//     Drive/Inputs/In/nState1 @bit 5 <-> DCM Status Channel 2/Status/Moving negative
//     Drive/Inputs/In/nState1 @bit 4 <-> DCM Status Channel 1/Status/Moving positive
//     Drive/Inputs/In/nState1 @bit 4 <-> DCM Status Channel 2/Status/Moving positive
//     Drive/Inputs/In/nState1 @bit 1 <-> DCM Status Channel 1/Status/Ready
//     Drive/Inputs/In/nState1 @bit 1 <-> DCM Status Channel 2/Status/Ready
//     Drive/Inputs/In/nState1 <-> DCM Status Channel 1/Status/Ready to enable
//     Drive/Inputs/In/nState1 <-> DCM Status Channel 2/Status/Ready to enable
//     Drive/Inputs/In/nState1 @bit 6 <-> DCM Status Channel 1/Status/Torque reduced
//     Drive/Inputs/In/nState1 @bit 6 <-> DCM Status Channel 2/Status/Torque reduced
//     Drive/Inputs/In/nState1 @bit 2 <-> DCM Status Channel 1/Status/Warning
//     Drive/Inputs/In/nState1 @bit 2 <-> DCM Status Channel 2/Status/Warning
//     Drive/Inputs/In/nState2 @bit 3 <-> DCM Status Channel 1/Status/Digital input 1
//     Drive/Inputs/In/nState2 @bit 4 <-> DCM Status Channel 1/Status/Digital input 2
//     Drive/Inputs/In/nState2 @bit 3 <-> DCM Status Channel 2/Status/Digital input 1
//     Drive/Inputs/In/nState2 @bit 4 <-> DCM Status Channel 2/Status/Digital input 2
//     Drive/Inputs/In/nState2 @bit 5 <-> DCM Status Channel 1/Status/Sync error
//     Drive/Inputs/In/nState2 @bit 5 <-> DCM Status Channel 2/Status/Sync error
//     Drive/Inputs/In/nState2 @bit 7 <-> DCM Status Channel 1/Status/TxPDO Toggle
//     Drive/Inputs/In/nState2 @bit 7 <-> DCM Status Channel 2/Status/TxPDO Toggle
//     Drive/Inputs/In/nState4 @bit 1 <-> WcState/InputToggle
//     Drive/Inputs/In/nState4 <-> WcState/WcState
//     Drive/Outputs/Out/nCtrl1 <-> DCM Control Channel 1/Control/Enable
//     Drive/Outputs/Out/nCtrl1 <-> DCM Control Channel 2/Control/Enable
//     Drive/Outputs/Out/nCtrl1 @bit 2 <-> DCM Control Channel 1/Control/Reduce torque
//     Drive/Outputs/Out/nCtrl1 @bit 2 <-> DCM Control Channel 2/Control/Reduce torque
//     Drive/Outputs/Out/nCtrl1 @bit 1 <-> DCM Control Channel 1/Control/Reset
//     Drive/Outputs/Out/nCtrl1 @bit 1 <-> DCM Control Channel 2/Control/Reset
//     Drive/Outputs/Out/nDataOut2[0] <-> DCM Velocity Channel 1/Velocity
//     Drive/Outputs/Out/nDataOut2[0] <-> DCM Velocity Channel 2/Velocity
//     Enc/Inputs/In/nDataIn1[0] <-> ENC Status compact Channel 1/Counter value
//     Enc/Inputs/In/nDataIn1[0] <-> ENC Status compact Channel 2/Counter value
//     Enc/Inputs/In/nDataIn2[0] <-> ENC Status compact Channel 1/Latch value
//     Enc/Inputs/In/nDataIn2[0] <-> ENC Status compact Channel 2/Latch value
//     Enc/Inputs/In/nState1 @bit 4 <-> ENC Status compact Channel 1/Status/Counter overflow
//     Enc/Inputs/In/nState1 @bit 4 <-> ENC Status compact Channel 2/Status/Counter overflow
//     Enc/Inputs/In/nState1 @bit 3 <-> ENC Status compact Channel 1/Status/Counter underflow
//     Enc/Inputs/In/nState1 @bit 3 <-> ENC Status compact Channel 2/Status/Counter underflow
//     Enc/Inputs/In/nState1 @bit 7 <-> ENC Status compact Channel 1/Status/Extrapolation stall
//     Enc/Inputs/In/nState1 @bit 7 <-> ENC Status compact Channel 2/Status/Extrapolation stall
//     Enc/Inputs/In/nState1 @bit 1 <-> ENC Status compact Channel 1/Status/Latch extern valid
//     Enc/Inputs/In/nState1 @bit 1 <-> ENC Status compact Channel 2/Status/Latch extern valid
//     Enc/Inputs/In/nState1 @bit 2 <-> ENC Status compact Channel 1/Status/Set counter done
//     Enc/Inputs/In/nState1 @bit 2 <-> ENC Status compact Channel 2/Status/Set counter done
//     Enc/Inputs/In/nState2 @bit 4 <-> ENC Status compact Channel 1/Status/Status of extern latch
//     Enc/Inputs/In/nState2 @bit 4 <-> ENC Status compact Channel 2/Status/Status of extern latch
//     Enc/Inputs/In/nState2 <-> ENC Status compact Channel 1/Status/Status of input A
//     Enc/Inputs/In/nState2 <-> ENC Status compact Channel 2/Status/Status of input A
//     Enc/Inputs/In/nState2 @bit 1 <-> ENC Status compact Channel 1/Status/Status of input B
//     Enc/Inputs/In/nState2 @bit 1 <-> ENC Status compact Channel 2/Status/Status of input B
//     Enc/Inputs/In/nState2 @bit 5 <-> ENC Status compact Channel 1/Status/Sync error
//     Enc/Inputs/In/nState2 @bit 5 <-> ENC Status compact Channel 2/Status/Sync error
//     Enc/Inputs/In/nState2 @bit 7 <-> ENC Status compact Channel 1/Status/TxPDO Toggle
//     Enc/Inputs/In/nState2 @bit 7 <-> ENC Status compact Channel 2/Status/TxPDO Toggle
//     Enc/Inputs/In/nState4 @bit 1 <-> WcState/InputToggle
//     Enc/Inputs/In/nState4 <-> WcState/WcState
//     Enc/Outputs/Out/nCtrl1 @bit 3 <-> ENC Control compact Channel 1/Control/Enable latch extern on negative edge
//     Enc/Outputs/Out/nCtrl1 @bit 3 <-> ENC Control compact Channel 2/Control/Enable latch extern on negative edge
//     Enc/Outputs/Out/nCtrl1 @bit 1 <-> ENC Control compact Channel 1/Control/Enable latch extern on positive edge
//     Enc/Outputs/Out/nCtrl1 @bit 1 <-> ENC Control compact Channel 2/Control/Enable latch extern on positive edge
//     Enc/Outputs/Out/nCtrl1 @bit 2 <-> ENC Control compact Channel 1/Control/Set counter
//     Enc/Outputs/Out/nCtrl1 @bit 2 <-> ENC Control compact Channel 2/Control/Set counter
//     Enc/Outputs/Out/nDataOut1[0] <-> ENC Control compact Channel 1/Set counter value
//     Enc/Outputs/Out/nDataOut1[0] <-> ENC Control compact Channel 2/Set counter value
//   (this object) <-> Device 1 (EtherCAT)/Power (EK1200)/PLC Junction 3 (EK1122)/X1 TMO FEE EC1 (EK1100)/TMO FEE EC1 E1 (EK1122)/X2-ST1K4-TEST (EK1100)/ST1K4-EL5042-E6
//     Enc/Inputs/In/nComState @bit 1 <-> WcState/InputToggle
//     Enc/Inputs/In/nComState <-> WcState/WcState
//     Enc/Inputs/In/nDataIn1 <-> FB Inputs Channel 1/Position
//     Enc/Inputs/In/nState1 @bit 12 <-> FB Inputs Channel 1/Status/Diag
//     Enc/Inputs/In/nState1 @bit 1 <-> FB Inputs Channel 1/Status/Error
//     Enc/Inputs/In/nState1 @bit 14 <-> FB Inputs Channel 1/Status/Input cycle counter
//     Enc/Inputs/In/nState1 @bit 2 <-> FB Inputs Channel 1/Status/Ready
//     Enc/Inputs/In/nState1 @bit 13 <-> FB Inputs Channel 1/Status/TxPDO State
//     Enc/Inputs/In/nState1 <-> FB Inputs Channel 1/Status/Warning
//   (this object) <-> Device 1 (EtherCAT)/Power (EK1200)/PLC Junction 3 (EK1122)/X1 TMO FEE EC1 (EK1100)/TMO FEE EC1 E1 (EK1122)/X2-ST1K4-TEST (EK1100)/ST1K4-EL7041-E4
//     Drive/Inputs/In/nState1 @bit 3 <-> STM Status/Status/Error
//     Drive/Inputs/In/nState1 @bit 5 <-> STM Status/Status/Moving negative
//     Drive/Inputs/In/nState1 @bit 4 <-> STM Status/Status/Moving positive
//     Drive/Inputs/In/nState1 @bit 1 <-> STM Status/Status/Ready
//     Drive/Inputs/In/nState1 <-> STM Status/Status/Ready to enable
//     Drive/Inputs/In/nState1 @bit 6 <-> STM Status/Status/Torque reduced
//     Drive/Inputs/In/nState1 @bit 2 <-> STM Status/Status/Warning
//     Drive/Inputs/In/nState2 @bit 3 <-> STM Status/Status/Digital input 1
//     Drive/Inputs/In/nState2 @bit 4 <-> STM Status/Status/Digital input 2
//     Drive/Inputs/In/nState2 @bit 5 <-> STM Status/Status/Sync error
//     Drive/Inputs/In/nState2 @bit 7 <-> STM Status/Status/TxPDO Toggle
//     Drive/Inputs/In/nState4 @bit 1 <-> WcState/InputToggle
//     Drive/Inputs/In/nState4 <-> WcState/WcState
//     Drive/Outputs/Out/nCtrl1 <-> STM Control/Control/Enable
//     Drive/Outputs/Out/nCtrl1 @bit 2 <-> STM Control/Control/Reduce torque
//     Drive/Outputs/Out/nCtrl1 @bit 1 <-> STM Control/Control/Reset
//     Drive/Outputs/Out/nDataOut2[0] <-> STM Velocity/Velocity
//   kfe_motion Instance <-> Device 1 (EtherCAT)/Power (EK1200)/PLC Junction 1 (EK1122)/X1 RTDSK0 (EK1100)/RTDSK0-EL2004
//     PlcTask Outputs/PRG_RTDSK0.bRTDSK0_SCRP_LED_01 <-> Channel 3/Output
//   kfe_motion Instance <-> Device 1 (EtherCAT)/Power (EK1200)/PLC Junction 1 (EK1122)/X1 RTDSK0 (EK1100)/RTDSK0-M2-EL7041
//     PlcTask Inputs/Main.M11.bLimitBackwardEnable <-> STM Status/Status/Digital input 2
//     PlcTask Inputs/Main.M11.bLimitForwardEnable <-> STM Status/Status/Digital input 1
//   kfe_motion Instance <-> Device 1 (EtherCAT)/Power (EK1200)/PLC Junction 1 (EK1122)/X1 RTDSK0 (EK1100)/RTDSK0-M3-EL7041
//     PlcTask Inputs/Main.M12.bLimitBackwardEnable <-> STM Status/Status/Digital input 2
//     PlcTask Inputs/Main.M12.bLimitForwardEnable <-> STM Status/Status/Digital input 1
//   kfe_motion Instance <-> Device 1 (EtherCAT)/Power (EK1200)/PLC Junction 1 (EK1122)/X1 RTDSK0 (EK1100)/RTDSK0-M4-EL7041
//     PlcTask Inputs/Main.M13.bLimitBackwardEnable <-> STM Status/Status/Digital input 2
//     PlcTask Inputs/Main.M13.bLimitForwardEnable <-> STM Status/Status/Digital input 1
//   kfe_motion Instance <-> Device 1 (EtherCAT)/Power (EK1200)/PLC Junction 1 (EK1122)/X1 RTDSK0 (EK1100)/RTDSK0-MPA-EL1008
//     PlcTask Inputs/PRG_RTDSK0.RTDSK0_MPA_01.i_xInsertedLS <-> Channel 1/Input
//     PlcTask Inputs/PRG_RTDSK0.RTDSK0_MPA_02.i_xInsertedLS <-> Channel 3/Input
//     PlcTask Inputs/PRG_RTDSK0.RTDSK0_MPA_03.i_xInsertedLS <-> Channel 5/Input
//     PlcTask Inputs/PRG_RTDSK0.RTDSK0_MPA_04.i_xInsertedLS <-> Channel 7/Input
//     PlcTask Inputs/PRG_RTDSK0.RTDSK0_MPA_01.i_xRetractedLS <-> Channel 2/Input
//     PlcTask Inputs/PRG_RTDSK0.RTDSK0_MPA_02.i_xRetractedLS <-> Channel 4/Input
//     PlcTask Inputs/PRG_RTDSK0.RTDSK0_MPA_03.i_xRetractedLS <-> Channel 6/Input
//     PlcTask Inputs/PRG_RTDSK0.RTDSK0_MPA_04.i_xRetractedLS <-> Channel 8/Input
//   kfe_motion Instance <-> Device 1 (EtherCAT)/Power (EK1200)/PLC Junction 1 (EK1122)/X1 RTDSK0 (EK1100)/RTDSK0-MPA-EL2008
//     PlcTask Outputs/PRG_RTDSK0.RTDSK0_MPA_01.q_xInsert_DO <-> Channel 1/Output
//     PlcTask Outputs/PRG_RTDSK0.RTDSK0_MPA_02.q_xInsert_DO <-> Channel 3/Output
//     PlcTask Outputs/PRG_RTDSK0.RTDSK0_MPA_03.q_xInsert_DO <-> Channel 5/Output
//     PlcTask Outputs/PRG_RTDSK0.RTDSK0_MPA_04.q_xInsert_DO <-> Channel 7/Output
//     PlcTask Outputs/PRG_RTDSK0.RTDSK0_MPA_01.q_xRetract_DO <-> Channel 2/Output
//     PlcTask Outputs/PRG_RTDSK0.RTDSK0_MPA_02.q_xRetract_DO <-> Channel 4/Output
//     PlcTask Outputs/PRG_RTDSK0.RTDSK0_MPA_03.q_xRetract_DO <-> Channel 6/Output
//     PlcTask Outputs/PRG_RTDSK0.RTDSK0_MPA_04.q_xRetract_DO <-> Channel 8/Output
//   kfe_motion Instance <-> Device 1 (EtherCAT)/Power (EK1200)/PLC Junction 1 (EK1122)/X2 IM1K0-XTES (EK1100)/IM1K0-EL1004
//     PlcTask Inputs/PRG_IM1K0_XTES.fbIM1K0.fbFlowSwitch.bFlowOk <-> Channel 2/Input
//     PlcTask Inputs/PRG_OTHER.fbPC1K0FlowSwitch.bFlowOk <-> Channel 1/Input
//     PlcTask Inputs/PRG_SL1K0_POWER.fbSL1K0.fbFlowSwitch.bFlowOk <-> Channel 3/Input
//   kfe_motion Instance <-> Device 1 (EtherCAT)/Power (EK1200)/PLC Junction 1 (EK1122)/X2 IM1K0-XTES (EK1100)/IM1K0-EL1088
//     PlcTask Inputs/Main.M2.bHome <-> Channel 2/Input
//     PlcTask Inputs/Main.M3.bHome <-> Channel 4/Input
//     PlcTask Inputs/PRG_IM1K0_XTES.fbIM1K0.bFocusEndBwd <-> Channel 4/Input
//     PlcTask Inputs/PRG_IM1K0_XTES.fbIM1K0.bFocusEndFwd <-> Channel 3/Input
//     PlcTask Inputs/PRG_IM1K0_XTES.fbIM1K0.bZoomEndBwd <-> Channel 2/Input
//     PlcTask Inputs/PRG_IM1K0_XTES.fbIM1K0.bZoomEndFwd <-> Channel 1/Input
//   kfe_motion Instance <-> Device 1 (EtherCAT)/Power (EK1200)/PLC Junction 1 (EK1122)/X2 IM1K0-XTES (EK1100)/IM1K0-EL2004
//     PlcTask Outputs/Main.M1.bBrakeRelease <-> Channel 1/Output
//     PlcTask Outputs/PRG_IM1K0_XTES.fbIM1K0.fbLED.bLEDPower <-> Channel 3/Output
//     PlcTask Outputs/PRG_IM1K0_XTES.fbIM1K0.fbOpal.bOpalPower <-> Channel 2/Output
//   kfe_motion Instance <-> Device 1 (EtherCAT)/Power (EK1200)/PLC Junction 1 (EK1122)/X2 IM1K0-XTES (EK1100)/IM1K0-EL3054
//     PlcTask Inputs/Main.M1.nRawEncoderINT <-> AI Standard Channel 1/Value
//   kfe_motion Instance <-> Device 1 (EtherCAT)/Power (EK1200)/PLC Junction 1 (EK1122)/X2 IM1K0-XTES (EK1100)/IM1K0-EL5101-01
//     PlcTask Inputs/Main.M2.nRawEncoderUINT <-> ENC Status compact/Counter value
//     PlcTask Inputs/Main.M3.nRawEncoderUINT <-> ENC Status compact/Counter value
//   kfe_motion Instance <-> Device 1 (EtherCAT)/Power (EK1200)/PLC Junction 1 (EK1122)/X2 IM1K0-XTES (EK1100)/IM1K0-EL6002
//     PlcTask Inputs/PRG_IM1K0_XTES.stEL6In/D[{0..21}] <-> COM TxPDO-Map Inputs Channel 1/Data In {0..21}  (22 links)
//     PlcTask Inputs/PRG_IM1K0_XTES.stEL6In/Status <-> COM TxPDO-Map Inputs Channel 1/Status
//     PlcTask Outputs/PRG_IM1K0_XTES.stEL6Out/Ctrl <-> COM RxPDO-Map Outputs Channel 1/Ctrl
//     PlcTask Outputs/PRG_IM1K0_XTES.stEL6Out/D[{0..21}] <-> COM RxPDO-Map Outputs Channel 1/Data Out {0..21}  (22 links)
//   kfe_motion Instance <-> Device 1 (EtherCAT)/Power (EK1200)/PLC Junction 1 (EK1122)/X2 IM1K0-XTES (EK1100)/IM1K0-EL7041
//     PlcTask Inputs/Main.M1.bLimitForwardEnable <-> STM Status/Status/Digital input 1
//   kfe_motion Instance <-> Device 1 (EtherCAT)/Power (EK1200)/PLC Junction 2 (EK1122)/X1 SL1K0-POWER (EK1100)/SL1K0-EL3054-E12
//     PlcTask Inputs/Main.M{18..21}.nRawEncoderINT <-> AI Standard Channel {1..4}/Value  (4 links)
//   kfe_motion Instance <-> Device 1 (EtherCAT)/Power (EK1200)/PLC Junction 2 (EK1122)/X1 SL1K0-POWER (EK1100)/SL1K0-EL3202-E6
//     PlcTask Inputs/PRG_SL1K0_POWER.fbSL1K0.RTD_South_1.bError <-> RTD Inputs Channel 1/Status/Error
//     PlcTask Inputs/PRG_SL1K0_POWER.fbSL1K0.RTD_South_2.bError <-> RTD Inputs Channel 2/Status/Error
//     PlcTask Inputs/PRG_SL1K0_POWER.fbSL1K0.RTD_South_1.bOverrange <-> RTD Inputs Channel 1/Status/Overrange
//     PlcTask Inputs/PRG_SL1K0_POWER.fbSL1K0.RTD_South_2.bOverrange <-> RTD Inputs Channel 2/Status/Overrange
//     PlcTask Inputs/PRG_SL1K0_POWER.fbSL1K0.RTD_South_1.bUnderrange <-> RTD Inputs Channel 1/Status/Underrange
//     PlcTask Inputs/PRG_SL1K0_POWER.fbSL1K0.RTD_South_2.bUnderrange <-> RTD Inputs Channel 2/Status/Underrange
//     PlcTask Inputs/PRG_SL1K0_POWER.fbSL1K0.RTD_South_1.iRaw <-> RTD Inputs Channel 1/Value
//     PlcTask Inputs/PRG_SL1K0_POWER.fbSL1K0.RTD_South_2.iRaw <-> RTD Inputs Channel 2/Value
//   kfe_motion Instance <-> Device 1 (EtherCAT)/Power (EK1200)/PLC Junction 2 (EK1122)/X1 SL1K0-POWER (EK1100)/SL1K0-EL3202-E7
//     PlcTask Inputs/PRG_SL1K0_POWER.fbSL1K0.RTD_TOP_1.bError <-> RTD Inputs Channel 1/Status/Error
//     PlcTask Inputs/PRG_SL1K0_POWER.fbSL1K0.RTD_TOP_2.bError <-> RTD Inputs Channel 2/Status/Error
//     PlcTask Inputs/PRG_SL1K0_POWER.fbSL1K0.RTD_TOP_1.bOverrange <-> RTD Inputs Channel 1/Status/Overrange
//     PlcTask Inputs/PRG_SL1K0_POWER.fbSL1K0.RTD_TOP_2.bOverrange <-> RTD Inputs Channel 2/Status/Overrange
//     PlcTask Inputs/PRG_SL1K0_POWER.fbSL1K0.RTD_TOP_1.bUnderrange <-> RTD Inputs Channel 1/Status/Underrange
//     PlcTask Inputs/PRG_SL1K0_POWER.fbSL1K0.RTD_TOP_2.bUnderrange <-> RTD Inputs Channel 2/Status/Underrange
//     PlcTask Inputs/PRG_SL1K0_POWER.fbSL1K0.RTD_TOP_1.iRaw <-> RTD Inputs Channel 1/Value
//     PlcTask Inputs/PRG_SL1K0_POWER.fbSL1K0.RTD_TOP_2.iRaw <-> RTD Inputs Channel 2/Value
//   kfe_motion Instance <-> Device 1 (EtherCAT)/Power (EK1200)/PLC Junction 2 (EK1122)/X1 SL1K0-POWER (EK1100)/SL1K0-EL3202-E8
//     PlcTask Inputs/PRG_SL1K0_POWER.fbSL1K0.RTD_North_1.bError <-> RTD Inputs Channel 1/Status/Error
//     PlcTask Inputs/PRG_SL1K0_POWER.fbSL1K0.RTD_North_2.bError <-> RTD Inputs Channel 2/Status/Error
//     PlcTask Inputs/PRG_SL1K0_POWER.fbSL1K0.RTD_North_1.bOverrange <-> RTD Inputs Channel 1/Status/Overrange
//     PlcTask Inputs/PRG_SL1K0_POWER.fbSL1K0.RTD_North_2.bOverrange <-> RTD Inputs Channel 2/Status/Overrange
//     PlcTask Inputs/PRG_SL1K0_POWER.fbSL1K0.RTD_North_1.bUnderrange <-> RTD Inputs Channel 1/Status/Underrange
//     PlcTask Inputs/PRG_SL1K0_POWER.fbSL1K0.RTD_North_2.bUnderrange <-> RTD Inputs Channel 2/Status/Underrange
//     PlcTask Inputs/PRG_SL1K0_POWER.fbSL1K0.RTD_North_1.iRaw <-> RTD Inputs Channel 1/Value
//     PlcTask Inputs/PRG_SL1K0_POWER.fbSL1K0.RTD_North_2.iRaw <-> RTD Inputs Channel 2/Value
//   kfe_motion Instance <-> Device 1 (EtherCAT)/Power (EK1200)/PLC Junction 2 (EK1122)/X1 SL1K0-POWER (EK1100)/SL1K0-EL3202-E9
//     PlcTask Inputs/PRG_SL1K0_POWER.fbSL1K0.RTD_Bottom_1.bError <-> RTD Inputs Channel 1/Status/Error
//     PlcTask Inputs/PRG_SL1K0_POWER.fbSL1K0.RTD_Bottom_2.bError <-> RTD Inputs Channel 2/Status/Error
//     PlcTask Inputs/PRG_SL1K0_POWER.fbSL1K0.RTD_Bottom_1.bOverrange <-> RTD Inputs Channel 1/Status/Overrange
//     PlcTask Inputs/PRG_SL1K0_POWER.fbSL1K0.RTD_Bottom_2.bOverrange <-> RTD Inputs Channel 2/Status/Overrange
//     PlcTask Inputs/PRG_SL1K0_POWER.fbSL1K0.RTD_Bottom_1.bUnderrange <-> RTD Inputs Channel 1/Status/Underrange
//     PlcTask Inputs/PRG_SL1K0_POWER.fbSL1K0.RTD_Bottom_2.bUnderrange <-> RTD Inputs Channel 2/Status/Underrange
//     PlcTask Inputs/PRG_SL1K0_POWER.fbSL1K0.RTD_Bottom_1.iRaw <-> RTD Inputs Channel 1/Value
//     PlcTask Inputs/PRG_SL1K0_POWER.fbSL1K0.RTD_Bottom_2.iRaw <-> RTD Inputs Channel 2/Value
//   kfe_motion Instance <-> Device 1 (EtherCAT)/Power (EK1200)/PLC Junction 2 (EK1122)/X1 SL1K0-POWER (EK1100)/SL1K0-EL7041-E1
//     PlcTask Inputs/Main.M18.bLimitBackwardEnable <-> STM Status/Status/Digital input 1
//     PlcTask Inputs/Main.M18.bLimitForwardEnable <-> STM Status/Status/Digital input 2
//   kfe_motion Instance <-> Device 1 (EtherCAT)/Power (EK1200)/PLC Junction 2 (EK1122)/X1 SL1K0-POWER (EK1100)/SL1K0-EL7041-E2
//     PlcTask Inputs/Main.M19.bLimitBackwardEnable <-> STM Status/Status/Digital input 1
//     PlcTask Inputs/Main.M19.bLimitForwardEnable <-> STM Status/Status/Digital input 2
//   kfe_motion Instance <-> Device 1 (EtherCAT)/Power (EK1200)/PLC Junction 2 (EK1122)/X1 SL1K0-POWER (EK1100)/SL1K0-EL7041-E4
//     PlcTask Inputs/Main.M20.bLimitBackwardEnable <-> STM Status/Status/Digital input 1
//     PlcTask Inputs/Main.M20.bLimitForwardEnable <-> STM Status/Status/Digital input 2
//   kfe_motion Instance <-> Device 1 (EtherCAT)/Power (EK1200)/PLC Junction 2 (EK1122)/X1 SL1K0-POWER (EK1100)/SL1K0-EL7041-E5
//     PlcTask Inputs/Main.M21.bLimitBackwardEnable <-> STM Status/Status/Digital input 1
//     PlcTask Inputs/Main.M21.bLimitForwardEnable <-> STM Status/Status/Digital input 2
//   kfe_motion Instance <-> Device 1 (EtherCAT)/Power (EK1200)/PLC Junction 2 (EK1122)/X2 SXR EC1 (EK1100)/EC1 E1 (EK1122)/X1 IM2K0-XTES (EK1100)/IM2K0-EL1088
//     PlcTask Inputs/Main.M6.bHome <-> Channel 2/Input
//     PlcTask Inputs/Main.M7.bHome <-> Channel 4/Input
//   kfe_motion Instance <-> Device 1 (EtherCAT)/Power (EK1200)/PLC Junction 2 (EK1122)/X2 SXR EC1 (EK1100)/EC1 E1 (EK1122)/X1 IM2K0-XTES (EK1100)/IM2K0-EL2004
//     PlcTask Outputs/Main.M5.bBrakeRelease <-> Channel 1/Output
//     PlcTask Outputs/PRG_IM2K0_XTES.fbIM2K0.fbGige.bGigePower <-> Channel 4/Output
//     PlcTask Outputs/PRG_IM2K0_XTES.fbIM2K0.fbLED.bLEDPower <-> Channel 3/Output
//   kfe_motion Instance <-> Device 1 (EtherCAT)/Power (EK1200)/PLC Junction 2 (EK1122)/X2 SXR EC1 (EK1100)/EC1 E1 (EK1122)/X1 IM2K0-XTES (EK1100)/IM2K0-EL5042
//     PlcTask Inputs/Main.M5.nRawEncoderULINT <-> FB Inputs Channel 1/Position
//   kfe_motion Instance <-> Device 1 (EtherCAT)/Power (EK1200)/PLC Junction 2 (EK1122)/X2 SXR EC1 (EK1100)/EC1 E1 (EK1122)/X1 IM2K0-XTES (EK1100)/IM2K0-EL7041
//     PlcTask Inputs/PRG_IM2K0_XTES.bDefectiveLimitSwitch <-> STM Status/Status/Digital input 1
//   kfe_motion Instance <-> Device 1 (EtherCAT)/Power (EK1200)/PLC Junction 2 (EK1122)/X2 SXR EC1 (EK1100)/EC1 E1 (EK1122)/X1 IM2K0-XTES (EK1100)/IM2K0-EL7342
//     PlcTask Inputs/Main.M6.nRawEncoderUINT <-> ENC Status compact Channel 1/Counter value
//     PlcTask Inputs/Main.M7.nRawEncoderUINT <-> ENC Status compact Channel 2/Counter value
//   kfe_motion Instance <-> Device 1 (EtherCAT)/Power (EK1200)/PLC Junction 2 (EK1122)/X2 SXR EC1 (EK1100)/EC1 E1 (EK1122)/X2 SL2K0-POWER (EK1100)/SL2K0-EL1004-E12
//     PlcTask Inputs/PRG_IM2K0_XTES.fbIM2K0.fbFlowSwitch.bFlowOk <-> Channel 1/Input
//     PlcTask Inputs/PRG_PF1K0_WFS.fbPF1K0.fbFlowSwitch.bFlowOk <-> Channel 1/Input
//     PlcTask Inputs/PRG_SL2K0_POWER.fbSL2K0.fbFlowSwitch.bFlowOk <-> Channel 1/Input
//   kfe_motion Instance <-> Device 1 (EtherCAT)/Power (EK1200)/PLC Junction 2 (EK1122)/X2 SXR EC1 (EK1100)/EC1 E1 (EK1122)/X2 SL2K0-POWER (EK1100)/SL2K0-EL3202-E10
//     PlcTask Inputs/PRG_SL2K0_POWER.fbSL2K0.RTD_Bottom_1.bError <-> RTD Inputs Channel 1/Status/Error
//     PlcTask Inputs/PRG_SL2K0_POWER.fbSL2K0.RTD_Bottom_1.iRaw <-> RTD Inputs Channel 1/Value
//     PlcTask Inputs/PRG_SL2K0_POWER.fbSL2K0.RTD_North_1.bError <-> RTD Inputs Channel 1/Status/Error
//     PlcTask Inputs/PRG_SL2K0_POWER.fbSL2K0.RTD_North_2.bError <-> RTD Inputs Channel 2/Status/Error
//     PlcTask Inputs/PRG_SL2K0_POWER.fbSL2K0.RTD_North_1.bOverrange <-> RTD Inputs Channel 1/Status/Overrange
//     PlcTask Inputs/PRG_SL2K0_POWER.fbSL2K0.RTD_North_2.bOverrange <-> RTD Inputs Channel 2/Status/Overrange
//     PlcTask Inputs/PRG_SL2K0_POWER.fbSL2K0.RTD_North_1.bUnderrange <-> RTD Inputs Channel 1/Status/Underrange
//     PlcTask Inputs/PRG_SL2K0_POWER.fbSL2K0.RTD_North_2.bUnderrange <-> RTD Inputs Channel 2/Status/Underrange
//     PlcTask Inputs/PRG_SL2K0_POWER.fbSL2K0.RTD_North_1.iRaw <-> RTD Inputs Channel 1/Value
//     PlcTask Inputs/PRG_SL2K0_POWER.fbSL2K0.RTD_North_2.iRaw <-> RTD Inputs Channel 2/Value
//   kfe_motion Instance <-> Device 1 (EtherCAT)/Power (EK1200)/PLC Junction 2 (EK1122)/X2 SXR EC1 (EK1100)/EC1 E1 (EK1122)/X2 SL2K0-POWER (EK1100)/SL2K0-EL3202-E11
//     PlcTask Inputs/PRG_SL2K0_POWER.fbSL2K0.RTD_Bottom_1.bOverrange <-> RTD Inputs Channel 1/Status/Overrange
//     PlcTask Inputs/PRG_SL2K0_POWER.fbSL2K0.RTD_Bottom_2.bOverrange <-> RTD Inputs Channel 2/Status/Overrange
//     PlcTask Inputs/PRG_SL2K0_POWER.fbSL2K0.RTD_Bottom_1.bUnderrange <-> RTD Inputs Channel 1/Status/Underrange
//     PlcTask Inputs/PRG_SL2K0_POWER.fbSL2K0.RTD_Bottom_2.bUnderrange <-> RTD Inputs Channel 2/Status/Underrange
//     PlcTask Inputs/PRG_SL2K0_POWER.fbSL2K0.RTD_Bottom_2.bError <-> RTD Inputs Channel 2/Status/Error
//     PlcTask Inputs/PRG_SL2K0_POWER.fbSL2K0.RTD_Bottom_2.iRaw <-> RTD Inputs Channel 2/Value
//   kfe_motion Instance <-> Device 1 (EtherCAT)/Power (EK1200)/PLC Junction 2 (EK1122)/X2 SXR EC1 (EK1100)/EC1 E1 (EK1122)/X2 SL2K0-POWER (EK1100)/SL2K0-EL3202-E8
//     PlcTask Inputs/PRG_SL2K0_POWER.fbSL2K0.RTD_South_1.bError <-> RTD Inputs Channel 1/Status/Error
//     PlcTask Inputs/PRG_SL2K0_POWER.fbSL2K0.RTD_South_2.bError <-> RTD Inputs Channel 2/Status/Error
//     PlcTask Inputs/PRG_SL2K0_POWER.fbSL2K0.RTD_South_1.bOverrange <-> RTD Inputs Channel 1/Status/Overrange
//     PlcTask Inputs/PRG_SL2K0_POWER.fbSL2K0.RTD_South_2.bOverrange <-> RTD Inputs Channel 2/Status/Overrange
//     PlcTask Inputs/PRG_SL2K0_POWER.fbSL2K0.RTD_South_1.bUnderrange <-> RTD Inputs Channel 1/Status/Underrange
//     PlcTask Inputs/PRG_SL2K0_POWER.fbSL2K0.RTD_South_2.bUnderrange <-> RTD Inputs Channel 2/Status/Underrange
//     PlcTask Inputs/PRG_SL2K0_POWER.fbSL2K0.RTD_South_1.iRaw <-> RTD Inputs Channel 1/Value
//     PlcTask Inputs/PRG_SL2K0_POWER.fbSL2K0.RTD_South_2.iRaw <-> RTD Inputs Channel 2/Value
//   kfe_motion Instance <-> Device 1 (EtherCAT)/Power (EK1200)/PLC Junction 2 (EK1122)/X2 SXR EC1 (EK1100)/EC1 E1 (EK1122)/X2 SL2K0-POWER (EK1100)/SL2K0-EL3202-E9
//     PlcTask Inputs/PRG_SL2K0_POWER.fbSL2K0.RTD_TOP_1.bError <-> RTD Inputs Channel 1/Status/Error
//     PlcTask Inputs/PRG_SL2K0_POWER.fbSL2K0.RTD_TOP_2.bError <-> RTD Inputs Channel 2/Status/Error
//     PlcTask Inputs/PRG_SL2K0_POWER.fbSL2K0.RTD_TOP_1.bOverrange <-> RTD Inputs Channel 1/Status/Overrange
//     PlcTask Inputs/PRG_SL2K0_POWER.fbSL2K0.RTD_TOP_2.bOverrange <-> RTD Inputs Channel 2/Status/Overrange
//     PlcTask Inputs/PRG_SL2K0_POWER.fbSL2K0.RTD_TOP_1.bUnderrange <-> RTD Inputs Channel 1/Status/Underrange
//     PlcTask Inputs/PRG_SL2K0_POWER.fbSL2K0.RTD_TOP_2.bUnderrange <-> RTD Inputs Channel 2/Status/Underrange
//     PlcTask Inputs/PRG_SL2K0_POWER.fbSL2K0.RTD_TOP_1.iRaw <-> RTD Inputs Channel 1/Value
//     PlcTask Inputs/PRG_SL2K0_POWER.fbSL2K0.RTD_TOP_2.iRaw <-> RTD Inputs Channel 2/Value
//   kfe_motion Instance <-> Device 1 (EtherCAT)/Power (EK1200)/PLC Junction 2 (EK1122)/X2 SXR EC1 (EK1100)/EC1 E1 (EK1122)/X2 SL2K0-POWER (EK1100)/SL2K0-EL5042-E2
//     PlcTask Inputs/Main.M22.nRawEncoderUINT <-> FB Inputs Channel 1/Position
//     PlcTask Inputs/Main.M23.nRawEncoderUINT <-> FB Inputs Channel 2/Position
//   kfe_motion Instance <-> Device 1 (EtherCAT)/Power (EK1200)/PLC Junction 2 (EK1122)/X2 SXR EC1 (EK1100)/EC1 E1 (EK1122)/X2 SL2K0-POWER (EK1100)/SL2K0-EL5042-E6
//     PlcTask Inputs/Main.M24.nRawEncoderUINT <-> FB Inputs Channel 1/Position
//     PlcTask Inputs/Main.M25.nRawEncoderUINT <-> FB Inputs Channel 2/Position
//   kfe_motion Instance <-> Device 1 (EtherCAT)/Power (EK1200)/PLC Junction 2 (EK1122)/X2 SXR EC1 (EK1100)/EC1 E1 (EK1122)/X2 SL2K0-POWER (EK1100)/SL2K0-EL7041-E1
//     PlcTask Inputs/Main.M22.bLimitBackwardEnable <-> STM Status/Status/Digital input 1
//     PlcTask Inputs/Main.M22.bLimitForwardEnable <-> STM Status/Status/Digital input 2
//   kfe_motion Instance <-> Device 1 (EtherCAT)/Power (EK1200)/PLC Junction 2 (EK1122)/X2 SXR EC1 (EK1100)/EC1 E1 (EK1122)/X2 SL2K0-POWER (EK1100)/SL2K0-EL7041-E3
//     PlcTask Inputs/Main.M23.bLimitBackwardEnable <-> STM Status/Status/Digital input 1
//     PlcTask Inputs/Main.M23.bLimitForwardEnable <-> STM Status/Status/Digital input 2
//   kfe_motion Instance <-> Device 1 (EtherCAT)/Power (EK1200)/PLC Junction 2 (EK1122)/X2 SXR EC1 (EK1100)/EC1 E1 (EK1122)/X2 SL2K0-POWER (EK1100)/SL2K0-EL7041-E5
//     PlcTask Inputs/Main.M24.bLimitBackwardEnable <-> STM Status/Status/Digital input 1
//     PlcTask Inputs/Main.M24.bLimitForwardEnable <-> STM Status/Status/Digital input 2
//   kfe_motion Instance <-> Device 1 (EtherCAT)/Power (EK1200)/PLC Junction 2 (EK1122)/X2 SXR EC1 (EK1100)/EC1 E1 (EK1122)/X2 SL2K0-POWER (EK1100)/SL2K0-EL7041-E7
//     PlcTask Inputs/Main.M25.bLimitBackwardEnable <-> STM Status/Status/Digital input 1
//     PlcTask Inputs/Main.M25.bLimitForwardEnable <-> STM Status/Status/Digital input 2
//   kfe_motion Instance <-> Device 1 (EtherCAT)/Power (EK1200)/PLC Junction 2 (EK1122)/X2 SXR EC1 (EK1100)/EC1 E2 (EK1122)/X1 PF1K0-WFS (EK1100)/PF1K0-EL2004
//     PlcTask Outputs/Main.M8.bBrakeRelease <-> Channel 1/Output
//   kfe_motion Instance <-> Device 1 (EtherCAT)/Power (EK1200)/PLC Junction 2 (EK1122)/X2 SXR EC1 (EK1100)/EC1 E2 (EK1122)/X1 PF1K0-WFS (EK1100)/PF1K0-EL3062
//     PlcTask Inputs/PRG_PF1K0_PM.fbPowerMeter.iVoltageINT <-> AI Standard Channel 1/Value
//   kfe_motion Instance <-> Device 1 (EtherCAT)/Power (EK1200)/PLC Junction 2 (EK1122)/X2 SXR EC1 (EK1100)/EC1 E2 (EK1122)/X1 PF1K0-WFS (EK1100)/PF1K0-EL3314
//     PlcTask Inputs/PRG_PF1K0_PM.fbPowerMeter.fbThermoCouple.bError <-> TC Inputs Channel 1/Status/Error
//     PlcTask Inputs/PRG_PF1K0_PM.fbPowerMeter.fbThermoCouple.bOverrange <-> TC Inputs Channel 1/Status/Overrange
//     PlcTask Inputs/PRG_PF1K0_PM.fbPowerMeter.fbThermoCouple.bUnderrange <-> TC Inputs Channel 1/Status/Underrange
//     PlcTask Inputs/PRG_PF1K0_PM.fbPowerMeter.fbThermoCouple.iRaw <-> TC Inputs Channel 1/Value
//     PlcTask Inputs/PRG_PF1K0_WFS.fbPF1K0.fbThermoCouple1.bError <-> TC Inputs Channel 1/Status/Error
//     PlcTask Inputs/PRG_PF1K0_WFS.fbPF1K0.fbThermoCouple2.bError <-> TC Inputs Channel 2/Status/Error
//     PlcTask Inputs/PRG_PF1K0_WFS.fbPF1K0.fbThermoCouple1.bOverrange <-> TC Inputs Channel 1/Status/Overrange
//     PlcTask Inputs/PRG_PF1K0_WFS.fbPF1K0.fbThermoCouple2.bOverrange <-> TC Inputs Channel 2/Status/Overrange
//     PlcTask Inputs/PRG_PF1K0_WFS.fbPF1K0.fbThermoCouple1.bUnderrange <-> TC Inputs Channel 1/Status/Underrange
//     PlcTask Inputs/PRG_PF1K0_WFS.fbPF1K0.fbThermoCouple2.bUnderrange <-> TC Inputs Channel 2/Status/Underrange
//     PlcTask Inputs/PRG_PF1K0_WFS.fbPF1K0.fbThermoCouple1.iRaw <-> TC Inputs Channel 1/Value
//     PlcTask Inputs/PRG_PF1K0_WFS.fbPF1K0.fbThermoCouple2.iRaw <-> TC Inputs Channel 2/Value
//   kfe_motion Instance <-> Device 1 (EtherCAT)/Power (EK1200)/PLC Junction 2 (EK1122)/X2 SXR EC1 (EK1100)/EC1 E2 (EK1122)/X1 PF1K0-WFS (EK1100)/PF1K0-EL5042
//     PlcTask Inputs/Main.M8.nRawEncoderULINT <-> FB Inputs Channel 2/Position
//     PlcTask Inputs/Main.M9.nRawEncoderULINT <-> FB Inputs Channel 1/Position
//   kfe_motion Instance <-> Device 1 (EtherCAT)/Power (EK1200)/PLC Junction 2 (EK1122)/X2 SXR EC1 (EK1100)/EC1 E2 (EK1122)/X1 PF1K0-WFS (EK1100)/PF1K0-EL7041-01
//     PlcTask Inputs/Main.M8.bLimitBackwardEnable <-> STM Status/Status/Digital input 2
//     PlcTask Inputs/Main.M8.bLimitForwardEnable <-> STM Status/Status/Digital input 1
//   kfe_motion Instance <-> Device 1 (EtherCAT)/Power (EK1200)/PLC Junction 2 (EK1122)/X2 SXR EC1 (EK1100)/EC1 E2 (EK1122)/X1 PF1K0-WFS (EK1100)/PF1K0-MPA-EL1004
//     PlcTask Inputs/PRG_PF1K0_PM.PF1K0_MPA_01.i_xInsertedLS <-> Channel 2/Input
//     PlcTask Inputs/PRG_PF1K0_PM.PF1K0_MPA_01.i_xRetractedLS <-> Channel 1/Input
//   kfe_motion Instance <-> Device 1 (EtherCAT)/Power (EK1200)/PLC Junction 2 (EK1122)/X2 SXR EC1 (EK1100)/EC1 E2 (EK1122)/X1 PF1K0-WFS (EK1100)/PF1K0-MPA-EL2004
//     PlcTask Outputs/PRG_PF1K0_PM.PF1K0_MPA_01.q_xInsert_DO <-> Channel 1/Output
//     PlcTask Outputs/PRG_PF1K0_PM.PF1K0_MPA_01.q_xRetract_DO <-> Channel 2/Output
//   kfe_motion Instance <-> Device 1 (EtherCAT)/Power (EK1200)/PLC Junction 2 (EK1122)/X2 SXR EC1 (EK1100)/EC1 E2 (EK1122)/X2 IM1K3-PPM (EK1100)/IM1K3-EL2004
//     PlcTask Outputs/Main.M4.bBrakeRelease <-> Channel 1/Output
//     PlcTask Outputs/PRG_IM1K3_PPM.fbIM1K3.fbGige.bGigePower <-> Channel 2/Output
//   kfe_motion Instance <-> Device 1 (EtherCAT)/Power (EK1200)/PLC Junction 2 (EK1122)/X2 SXR EC1 (EK1100)/EC1 E2 (EK1122)/X2 IM1K3-PPM (EK1100)/IM1K3-EL3062
//     PlcTask Inputs/PRG_IM1K3_PPM.fbIM1K3.fbPowerMeter.iVoltageINT <-> AI Standard Channel 1/Value
//   kfe_motion Instance <-> Device 1 (EtherCAT)/Power (EK1200)/PLC Junction 2 (EK1122)/X2 SXR EC1 (EK1100)/EC1 E2 (EK1122)/X2 IM1K3-PPM (EK1100)/IM1K3-EL3314
//     PlcTask Inputs/PRG_IM1K3_PPM.fbIM1K3.fbPowerMeter.fbThermoCouple.bError <-> TC Inputs Channel 1/Status/Error
//     PlcTask Inputs/PRG_IM1K3_PPM.fbIM1K3.fbPowerMeter.fbThermoCouple.bOverrange <-> TC Inputs Channel 1/Status/Overrange
//     PlcTask Inputs/PRG_IM1K3_PPM.fbIM1K3.fbPowerMeter.fbThermoCouple.bUnderrange <-> TC Inputs Channel 1/Status/Underrange
//     PlcTask Inputs/PRG_IM1K3_PPM.fbIM1K3.fbPowerMeter.fbThermoCouple.iRaw <-> TC Inputs Channel 1/Value
//     PlcTask Inputs/PRG_IM1K3_PPM.fbIM1K3.fbYagThermoCouple.bError <-> TC Inputs Channel 2/Status/Error
//     PlcTask Inputs/PRG_IM1K3_PPM.fbIM1K3.fbYagThermoCouple.bOverrange <-> TC Inputs Channel 2/Status/Overrange
//     PlcTask Inputs/PRG_IM1K3_PPM.fbIM1K3.fbYagThermoCouple.bUnderrange <-> TC Inputs Channel 2/Status/Underrange
//     PlcTask Inputs/PRG_IM1K3_PPM.fbIM1K3.fbYagThermoCouple.iRaw <-> TC Inputs Channel 2/Value
//   kfe_motion Instance <-> Device 1 (EtherCAT)/Power (EK1200)/PLC Junction 2 (EK1122)/X2 SXR EC1 (EK1100)/EC1 E2 (EK1122)/X2 IM1K3-PPM (EK1100)/IM1K3-EL4004
//     PlcTask Outputs/PRG_IM1K3_PPM.fbIM1K3.fbGige.iIlluminatorINT <-> AO Outputs Channel 1/Analog output
//   kfe_motion Instance <-> Device 1 (EtherCAT)/Power (EK1200)/PLC Junction 2 (EK1122)/X2 SXR EC1 (EK1100)/EC1 E2 (EK1122)/X2 IM1K3-PPM (EK1100)/IM1K3-EL5042
//     PlcTask Inputs/Main.M4.nRawEncoderULINT <-> FB Inputs Channel 1/Position
//   kfe_motion Instance <-> Device 1 (EtherCAT)/Power (EK1200)/PLC Junction 2 (EK1122)/X2 SXR EC1 (EK1100)/EC1 E2 (EK1122)/X2 IM1K3-PPM (EK1100)/IM1K3-EL7041
//     PlcTask Inputs/Main.M4.bLimitBackwardEnable <-> STM Status/Status/Digital input 2
//     PlcTask Inputs/Main.M4.bLimitForwardEnable <-> STM Status/Status/Digital input 1
//   kfe_motion Instance <-> Device 1 (EtherCAT)/Power (EK1200)/PLC Junction 3 (EK1122)/X1 TMO FEE EC1 (EK1100)/TMO FEE EC1 E1 (EK1122)/X1 IM1K4-XTES (EK1100)/IM1K4-EL1088-E5
//     PlcTask Inputs/Main.M31.bHome <-> Channel 2/Input
//     PlcTask Inputs/Main.M32.bHome <-> Channel 4/Input
//     PlcTask Inputs/PRG_IM1K4_XTES.fbIM1K4.bFocusEndBwd <-> Channel 4/Input
//     PlcTask Inputs/PRG_IM1K4_XTES.fbIM1K4.bFocusEndFwd <-> Channel 3/Input
//     PlcTask Inputs/PRG_IM1K4_XTES.fbIM1K4.bZoomEndBwd <-> Channel 2/Input
//     PlcTask Inputs/PRG_IM1K4_XTES.fbIM1K4.bZoomEndFwd <-> Channel 1/Input
//   kfe_motion Instance <-> Device 1 (EtherCAT)/Power (EK1200)/PLC Junction 3 (EK1122)/X1 TMO FEE EC1 (EK1100)/TMO FEE EC1 E1 (EK1122)/X1 IM1K4-XTES (EK1100)/IM1K4-EL2004-E2
//     PlcTask Outputs/Main.M30.bBrakeRelease <-> Channel 1/Output
//     PlcTask Outputs/PRG_IM1K4_XTES.bIM1K4_SCRP_LED_01 <-> Channel 4/Output
//     PlcTask Outputs/PRG_IM1K4_XTES.fbIM1K4.fbLED.bLEDPower <-> Channel 3/Output
//     PlcTask Outputs/PRG_IM1K4_XTES.fbIM1K4.fbOpal.bOpalPower <-> Channel 2/Output
//   kfe_motion Instance <-> Device 1 (EtherCAT)/Power (EK1200)/PLC Junction 3 (EK1122)/X1 TMO FEE EC1 (EK1100)/TMO FEE EC1 E1 (EK1122)/X1 IM1K4-XTES (EK1100)/IM1K4-EL5042-E3
//     PlcTask Inputs/Main.M30.nRawEncoderULINT <-> FB Inputs Channel 1/Position
//   kfe_motion Instance <-> Device 1 (EtherCAT)/Power (EK1200)/PLC Junction 3 (EK1122)/X1 TMO FEE EC1 (EK1100)/TMO FEE EC1 E1 (EK1122)/X1 IM1K4-XTES (EK1100)/IM1K4-EL6002-E6
//     PlcTask Inputs/PRG_IM1K4_XTES.stEL6In/D[{0..21}] <-> COM TxPDO-Map Inputs Channel 1/Data In {0..21}  (22 links)
//     PlcTask Inputs/PRG_IM1K4_XTES.stEL6In/Status <-> COM TxPDO-Map Inputs Channel 1/Status
//     PlcTask Outputs/PRG_IM1K4_XTES.stEL6Out/Ctrl <-> COM RxPDO-Map Outputs Channel 1/Ctrl
//     PlcTask Outputs/PRG_IM1K4_XTES.stEL6Out/D[{0..21}] <-> COM RxPDO-Map Outputs Channel 1/Data Out {0..21}  (22 links)
//   kfe_motion Instance <-> Device 1 (EtherCAT)/Power (EK1200)/PLC Junction 3 (EK1122)/X1 TMO FEE EC1 (EK1100)/TMO FEE EC1 E1 (EK1122)/X1 IM1K4-XTES (EK1100)/IM1K4-EL7041-E1
//     PlcTask Inputs/Main.M30.bLimitForwardEnable <-> STM Status/Status/Digital input 1
//   kfe_motion Instance <-> Device 1 (EtherCAT)/Power (EK1200)/PLC Junction 3 (EK1122)/X1 TMO FEE EC1 (EK1100)/TMO FEE EC1 E1 (EK1122)/X1 IM1K4-XTES (EK1100)/IM1K4-EL7342-E4
//     PlcTask Inputs/Main.M31.nRawEncoderUINT <-> ENC Status compact Channel 1/Counter value
//     PlcTask Inputs/Main.M32.nRawEncoderUINT <-> ENC Status compact Channel 2/Counter value
//   kfe_motion Instance <-> Device 1 (EtherCAT)/Power (EK1200)/PLC Junction 3 (EK1122)/X1 TMO FEE EC1 (EK1100)/TMO FEE EC1 E1 (EK1122)/X2-ST1K4-TEST (EK1100)/ST1K4-EL1004-E5
//     PlcTask Inputs/PRG_IM1K3_PPM.fbIM1K3.fbFlowSwitch.bFlowOk <-> Channel 3/Input
//     PlcTask Inputs/PRG_IM1K4_XTES.fbIM1K4.fbFlowSwitch.bFlowOk <-> Channel 2/Input
//     PlcTask Inputs/PRG_OTHER.fbPC1K4FlowSwitch.bFlowOk <-> Channel 2/Input
//     PlcTask Inputs/PRG_ST1K4_TEST.fbFlowSwitch.bFlowOk <-> Channel 1/Input
//   kfe_motion Instance <-> Device 1 (EtherCAT)/Power (EK1200)/PLC Junction 3 (EK1122)/X1 TMO FEE EC1 (EK1100)/TMO FEE EC1 E1 (EK1122)/X2-ST1K4-TEST (EK1100)/ST1K4-EL2202-E3
//     PlcTask Outputs/Main.M33.bBrakeRelease <-> Channel 1/Output
//   kfe_motion Instance <-> Device 1 (EtherCAT)/Power (EK1200)/PLC Junction 3 (EK1122)/X1 TMO FEE EC1 (EK1100)/TMO FEE EC1 E1 (EK1122)/X2-ST1K4-TEST (EK1100)/ST1K4-EL5042-E6
//     PlcTask Inputs/Main.M33.nRawEncoderULINT <-> FB Inputs Channel 1/Position
//     PlcTask Inputs/PRG_ST1K4_TEST.nRawEncoderULINT <-> FB Inputs Channel 1/Position
//   kfe_motion Instance <-> Device 1 (EtherCAT)/Power (EK1200)/PLC Junction 3 (EK1122)/X1 TMO FEE EC1 (EK1100)/TMO FEE EC1 E1 (EK1122)/X2-ST1K4-TEST (EK1100)/ST1K4-EL7041-E4
//     PlcTask Inputs/Main.M33.bLimitBackwardEnable <-> STM Status/Status/Digital input 2
//     PlcTask Inputs/Main.M33.bLimitForwardEnable <-> STM Status/Status/Digital input 1
//   kfe_motion Instance <-> Device 1 (EtherCAT)/Power (EK1200)/PLC Junction 3 (EK1122)/X1 TMO FEE EC1 (EK1100)/TMO FEE EC1 E2 (EK1122)/X1 AT1K4-SOLID (EK1100)/AT1K4-EL3202-01
//     PlcTask Inputs/PRG_AT1K4_SOLID.fbStage4.fbRTD_1.bError <-> RTD Inputs Channel 1/Status/Error
//     PlcTask Inputs/PRG_AT1K4_SOLID.fbStage4.fbRTD_2.bError <-> RTD Inputs Channel 2/Status/Error
//     PlcTask Inputs/PRG_AT1K4_SOLID.fbStage4.fbRTD_1.bOverrange <-> RTD Inputs Channel 1/Status/Overrange
//     PlcTask Inputs/PRG_AT1K4_SOLID.fbStage4.fbRTD_2.bOverrange <-> RTD Inputs Channel 2/Status/Overrange
//     PlcTask Inputs/PRG_AT1K4_SOLID.fbStage4.fbRTD_1.bUnderrange <-> RTD Inputs Channel 1/Status/Underrange
//     PlcTask Inputs/PRG_AT1K4_SOLID.fbStage4.fbRTD_2.bUnderrange <-> RTD Inputs Channel 2/Status/Underrange
//     PlcTask Inputs/PRG_AT1K4_SOLID.fbStage4.fbRTD_1.iRaw <-> RTD Inputs Channel 1/Value
//     PlcTask Inputs/PRG_AT1K4_SOLID.fbStage4.fbRTD_2.iRaw <-> RTD Inputs Channel 2/Value
//   kfe_motion Instance <-> Device 1 (EtherCAT)/Power (EK1200)/PLC Junction 3 (EK1122)/X1 TMO FEE EC1 (EK1100)/TMO FEE EC1 E2 (EK1122)/X1 AT1K4-SOLID (EK1100)/AT1K4-EL3202-02
//     PlcTask Inputs/PRG_AT1K4_SOLID.fbStage3.fbRTD_1.bError <-> RTD Inputs Channel 1/Status/Error
//     PlcTask Inputs/PRG_AT1K4_SOLID.fbStage3.fbRTD_2.bError <-> RTD Inputs Channel 2/Status/Error
//     PlcTask Inputs/PRG_AT1K4_SOLID.fbStage3.fbRTD_1.bOverrange <-> RTD Inputs Channel 1/Status/Overrange
//     PlcTask Inputs/PRG_AT1K4_SOLID.fbStage3.fbRTD_2.bOverrange <-> RTD Inputs Channel 2/Status/Overrange
//     PlcTask Inputs/PRG_AT1K4_SOLID.fbStage3.fbRTD_1.bUnderrange <-> RTD Inputs Channel 1/Status/Underrange
//     PlcTask Inputs/PRG_AT1K4_SOLID.fbStage3.fbRTD_2.bUnderrange <-> RTD Inputs Channel 2/Status/Underrange
//     PlcTask Inputs/PRG_AT1K4_SOLID.fbStage3.fbRTD_1.iRaw <-> RTD Inputs Channel 1/Value
//     PlcTask Inputs/PRG_AT1K4_SOLID.fbStage3.fbRTD_2.iRaw <-> RTD Inputs Channel 2/Value
//   kfe_motion Instance <-> Device 1 (EtherCAT)/Power (EK1200)/PLC Junction 3 (EK1122)/X1 TMO FEE EC1 (EK1100)/TMO FEE EC1 E2 (EK1122)/X1 AT1K4-SOLID (EK1100)/AT1K4-EL3202-03
//     PlcTask Inputs/PRG_AT1K4_SOLID.fbStage2.fbRTD_1.bError <-> RTD Inputs Channel 1/Status/Error
//     PlcTask Inputs/PRG_AT1K4_SOLID.fbStage2.fbRTD_2.bError <-> RTD Inputs Channel 2/Status/Error
//     PlcTask Inputs/PRG_AT1K4_SOLID.fbStage2.fbRTD_1.bOverrange <-> RTD Inputs Channel 1/Status/Overrange
//     PlcTask Inputs/PRG_AT1K4_SOLID.fbStage2.fbRTD_2.bOverrange <-> RTD Inputs Channel 2/Status/Overrange
//     PlcTask Inputs/PRG_AT1K4_SOLID.fbStage2.fbRTD_1.bUnderrange <-> RTD Inputs Channel 1/Status/Underrange
//     PlcTask Inputs/PRG_AT1K4_SOLID.fbStage2.fbRTD_2.bUnderrange <-> RTD Inputs Channel 2/Status/Underrange
//     PlcTask Inputs/PRG_AT1K4_SOLID.fbStage2.fbRTD_1.iRaw <-> RTD Inputs Channel 1/Value
//     PlcTask Inputs/PRG_AT1K4_SOLID.fbStage2.fbRTD_2.iRaw <-> RTD Inputs Channel 2/Value
//   kfe_motion Instance <-> Device 1 (EtherCAT)/Power (EK1200)/PLC Junction 3 (EK1122)/X1 TMO FEE EC1 (EK1100)/TMO FEE EC1 E2 (EK1122)/X1 AT1K4-SOLID (EK1100)/AT1K4-EL3202-04
//     PlcTask Inputs/PRG_AT1K4_SOLID.fbStage1.fbRTD_1.bError <-> RTD Inputs Channel 1/Status/Error
//     PlcTask Inputs/PRG_AT1K4_SOLID.fbStage1.fbRTD_2.bError <-> RTD Inputs Channel 2/Status/Error
//     PlcTask Inputs/PRG_AT1K4_SOLID.fbStage1.fbRTD_1.bOverrange <-> RTD Inputs Channel 1/Status/Overrange
//     PlcTask Inputs/PRG_AT1K4_SOLID.fbStage1.fbRTD_2.bOverrange <-> RTD Inputs Channel 2/Status/Overrange
//     PlcTask Inputs/PRG_AT1K4_SOLID.fbStage1.fbRTD_1.bUnderrange <-> RTD Inputs Channel 1/Status/Underrange
//     PlcTask Inputs/PRG_AT1K4_SOLID.fbStage1.fbRTD_2.bUnderrange <-> RTD Inputs Channel 2/Status/Underrange
//     PlcTask Inputs/PRG_AT1K4_SOLID.fbStage1.fbRTD_1.iRaw <-> RTD Inputs Channel 1/Value
//     PlcTask Inputs/PRG_AT1K4_SOLID.fbStage1.fbRTD_2.iRaw <-> RTD Inputs Channel 2/Value
//   kfe_motion Instance <-> Device 1 (EtherCAT)/Power (EK1200)/PLC Junction 3 (EK1122)/X1 TMO FEE EC1 (EK1100)/TMO FEE EC1 E2 (EK1122)/X1 AT1K4-SOLID (EK1100)/AT1K4-EL5042-01
//     PlcTask Inputs/Main.M28.nRawEncoderULINT <-> FB Inputs Channel 2/Position
//     PlcTask Inputs/Main.M29.nRawEncoderULINT <-> FB Inputs Channel 1/Position
//   kfe_motion Instance <-> Device 1 (EtherCAT)/Power (EK1200)/PLC Junction 3 (EK1122)/X1 TMO FEE EC1 (EK1100)/TMO FEE EC1 E2 (EK1122)/X1 AT1K4-SOLID (EK1100)/AT1K4-EL5042-02
//     PlcTask Inputs/Main.M26.nRawEncoderULINT <-> FB Inputs Channel 2/Position
//     PlcTask Inputs/Main.M27.nRawEncoderULINT <-> FB Inputs Channel 1/Position
//   kfe_motion Instance <-> Device 1 (EtherCAT)/Power (EK1200)/PLC Junction 3 (EK1122)/X1 TMO FEE EC1 (EK1100)/TMO FEE EC1 E2 (EK1122)/X1 AT1K4-SOLID (EK1100)/AT1K4-EL7047-01
//     PlcTask Inputs/Main.M29.bLimitBackwardEnable <-> STM Status/Status/Digital input 2
//     PlcTask Inputs/Main.M29.bLimitForwardEnable <-> STM Status/Status/Digital input 1
//   kfe_motion Instance <-> Device 1 (EtherCAT)/Power (EK1200)/PLC Junction 3 (EK1122)/X1 TMO FEE EC1 (EK1100)/TMO FEE EC1 E2 (EK1122)/X1 AT1K4-SOLID (EK1100)/AT1K4-EL7047-02
//     PlcTask Inputs/Main.M28.bLimitBackwardEnable <-> STM Status/Status/Digital input 2
//     PlcTask Inputs/Main.M28.bLimitForwardEnable <-> STM Status/Status/Digital input 1
//   kfe_motion Instance <-> Device 1 (EtherCAT)/Power (EK1200)/PLC Junction 3 (EK1122)/X1 TMO FEE EC1 (EK1100)/TMO FEE EC1 E2 (EK1122)/X1 AT1K4-SOLID (EK1100)/AT1K4-EL7047-03
//     PlcTask Inputs/Main.M27.bLimitBackwardEnable <-> STM Status/Status/Digital input 2
//     PlcTask Inputs/Main.M27.bLimitForwardEnable <-> STM Status/Status/Digital input 1
//   kfe_motion Instance <-> Device 1 (EtherCAT)/Power (EK1200)/PLC Junction 3 (EK1122)/X1 TMO FEE EC1 (EK1100)/TMO FEE EC1 E2 (EK1122)/X1 AT1K4-SOLID (EK1100)/AT1K4-EL7047-04
//     PlcTask Inputs/Main.M26.bLimitBackwardEnable <-> STM Status/Status/Digital input 2
//     PlcTask Inputs/Main.M26.bLimitForwardEnable <-> STM Status/Status/Digital input 1
//   kfe_motion Instance <-> Device 1 (EtherCAT)/Power (EK1200)/PMPS_FFO
//     PlcTask Outputs/GVL.fbFastFaultOutput1.q_xFastFaultOut <-> Channel 1/Output
//     PlcTask Outputs/GVL.fbFastFaultOutput2.q_xFastFaultOut <-> Channel 2/Output
//   kfe_motion Instance <-> Device 1 (EtherCAT)/Power (EK1200)/PMPS_PRE
//     PlcTask Inputs/PRG_3_PMPS_POST.fbArbiterIO.i_stCurrentBP <-> IO Inputs/CurrentBP
//     PlcTask Inputs/PRG_3_PMPS_POST.fbArbiterIO.xTxPDO_state <-> SYNC Inputs/TxPDO state
//     PlcTask Inputs/PRG_3_PMPS_POST.fbArbiterIO.xTxPDO_toggle <-> SYNC Inputs/TxPDO toggle
//     PlcTask Inputs/PRG_SL1K0_POWER.fbSL1K0.AptArrayReq <-> IO Inputs/AptArrayReq[1]
//     PlcTask Inputs/PRG_SL2K0_POWER.fbSL2K0.AptArrayReq <-> IO Inputs/AptArrayReq[2]
//     PlcTask Outputs/GVL.PMPS_ST1K4_Y_ENC <-> IO Outputs/ST1K4_Y_ENC
//     PlcTask Outputs/PRG_3_PMPS_POST.fbArbiterIO.q_stRequestedBP <-> IO Outputs/RequestedBP
//     PlcTask Outputs/PRG_SL1K0_POWER.fbSL1K0.AptArrayStatus <-> IO Outputs/AptArrayStatus[1]
//     PlcTask Outputs/PRG_SL2K0_POWER.fbSL2K0.AptArrayStatus <-> IO Outputs/AptArrayStatus[2]
//   kfe_motion Instance <-> NC-Task 1 SAF/Axes/Axis 1 IM1K0-XTES-MMS
//     PlcTask Inputs/Main.M1.Axis.NcToPlc <-> Outputs/ToPlc
//     PlcTask Outputs/Main.M1.Axis.PlcToNc <-> Inputs/FromPlc
//   kfe_motion Instance <-> NC-Task 1 SAF/Axes/Axis 10
//     PlcTask Inputs/Main.M10.Axis.NcToPlc <-> Outputs/ToPlc
//     PlcTask Outputs/Main.M10.Axis.PlcToNc <-> Inputs/FromPlc
//   kfe_motion Instance <-> NC-Task 1 SAF/Axes/Axis 11-SCPR-Z
//     PlcTask Inputs/Main.M11.Axis.NcToPlc <-> Outputs/ToPlc
//     PlcTask Outputs/Main.M11.Axis.PlcToNc <-> Inputs/FromPlc
//   kfe_motion Instance <-> NC-Task 1 SAF/Axes/Axis 12-SCRP-X
//     PlcTask Inputs/Main.M12.Axis.NcToPlc <-> Outputs/ToPlc
//     PlcTask Outputs/Main.M12.Axis.PlcToNc <-> Inputs/FromPlc
//   kfe_motion Instance <-> NC-Task 1 SAF/Axes/Axis 13-SCRP-Y
//     PlcTask Inputs/Main.M13.Axis.NcToPlc <-> Outputs/ToPlc
//     PlcTask Outputs/Main.M13.Axis.PlcToNc <-> Inputs/FromPlc
//   kfe_motion Instance <-> NC-Task 1 SAF/Axes/Axis 14
//     PlcTask Inputs/Main.M14.Axis.NcToPlc <-> Outputs/ToPlc
//     PlcTask Outputs/Main.M14.Axis.PlcToNc <-> Inputs/FromPlc
//   kfe_motion Instance <-> NC-Task 1 SAF/Axes/Axis 15
//     PlcTask Inputs/Main.M15.Axis.NcToPlc <-> Outputs/ToPlc
//     PlcTask Outputs/Main.M15.Axis.PlcToNc <-> Inputs/FromPlc
//   kfe_motion Instance <-> NC-Task 1 SAF/Axes/Axis 16
//     PlcTask Inputs/Main.M16.Axis.NcToPlc <-> Outputs/ToPlc
//     PlcTask Outputs/Main.M16.Axis.PlcToNc <-> Inputs/FromPlc
//   kfe_motion Instance <-> NC-Task 1 SAF/Axes/Axis 17
//     PlcTask Inputs/Main.M17.Axis.NcToPlc <-> Outputs/ToPlc
//     PlcTask Outputs/Main.M17.Axis.PlcToNc <-> Inputs/FromPlc
//   kfe_motion Instance <-> NC-Task 1 SAF/Axes/Axis 2 IM1K0-XTES-CLZ
//     PlcTask Inputs/Main.M2.Axis.NcToPlc <-> Outputs/ToPlc
//     PlcTask Outputs/Main.M2.Axis.PlcToNc <-> Inputs/FromPlc
//   kfe_motion Instance <-> NC-Task 1 SAF/Axes/Axis 26 AT1K4-SOLID-01 MMS-01
//     PlcTask Inputs/Main.M26.Axis.NcToPlc <-> Outputs/ToPlc
//     PlcTask Outputs/Main.M26.Axis.PlcToNc <-> Inputs/FromPlc
//   kfe_motion Instance <-> NC-Task 1 SAF/Axes/Axis 27 AT1K4-SOLID-02 MMS-02
//     PlcTask Inputs/Main.M27.Axis.NcToPlc <-> Outputs/ToPlc
//     PlcTask Outputs/Main.M27.Axis.PlcToNc <-> Inputs/FromPlc
//   kfe_motion Instance <-> NC-Task 1 SAF/Axes/Axis 28 AT1K4-SOLID-03 MMS-03
//     PlcTask Inputs/Main.M28.Axis.NcToPlc <-> Outputs/ToPlc
//     PlcTask Outputs/Main.M28.Axis.PlcToNc <-> Inputs/FromPlc
//   kfe_motion Instance <-> NC-Task 1 SAF/Axes/Axis 29 AT1K4-SOLID-04 MMS-04
//     PlcTask Inputs/Main.M29.Axis.NcToPlc <-> Outputs/ToPlc
//     PlcTask Outputs/Main.M29.Axis.PlcToNc <-> Inputs/FromPlc
//   kfe_motion Instance <-> NC-Task 1 SAF/Axes/Axis 3 IM1K0-XTES-CLF
//     PlcTask Inputs/Main.M3.Axis.NcToPlc <-> Outputs/ToPlc
//     PlcTask Outputs/Main.M3.Axis.PlcToNc <-> Inputs/FromPlc
//   kfe_motion Instance <-> NC-Task 1 SAF/Axes/Axis 30 IM1K4-XTES-MMS
//     PlcTask Inputs/Main.M30.Axis.NcToPlc <-> Outputs/ToPlc
//     PlcTask Outputs/Main.M30.Axis.PlcToNc <-> Inputs/FromPlc
//   kfe_motion Instance <-> NC-Task 1 SAF/Axes/Axis 31 IM1K4-XTES-CLZ
//     PlcTask Inputs/Main.M31.Axis.NcToPlc <-> Outputs/ToPlc
//     PlcTask Outputs/Main.M31.Axis.PlcToNc <-> Inputs/FromPlc
//   kfe_motion Instance <-> NC-Task 1 SAF/Axes/Axis 32 IM1K4-XTES-CLF
//     PlcTask Inputs/Main.M32.Axis.NcToPlc <-> Outputs/ToPlc
//     PlcTask Outputs/Main.M32.Axis.PlcToNc <-> Inputs/FromPlc
//   kfe_motion Instance <-> NC-Task 1 SAF/Axes/Axis 4 IM1K3-PPM-MMS
//     PlcTask Inputs/Main.M4.Axis.NcToPlc <-> Outputs/ToPlc
//     PlcTask Outputs/Main.M4.Axis.PlcToNc <-> Inputs/FromPlc
//   kfe_motion Instance <-> NC-Task 1 SAF/Axes/Axis 5 IM2K0-XTES-MMS
//     PlcTask Inputs/Main.M5.Axis.NcToPlc <-> Outputs/ToPlc
//     PlcTask Outputs/Main.M5.Axis.PlcToNc <-> Inputs/FromPlc
//   kfe_motion Instance <-> NC-Task 1 SAF/Axes/Axis 6 IM2K0-XTES-CLZ (Removed)
//     PlcTask Inputs/Main.M6.Axis.NcToPlc <-> Outputs/ToPlc
//     PlcTask Outputs/Main.M6.Axis.PlcToNc <-> Inputs/FromPlc
//   kfe_motion Instance <-> NC-Task 1 SAF/Axes/Axis 7 IM2K0-XTES-CLF (Removed)
//     PlcTask Inputs/Main.M7.Axis.NcToPlc <-> Outputs/ToPlc
//     PlcTask Outputs/Main.M7.Axis.PlcToNc <-> Inputs/FromPlc
//   kfe_motion Instance <-> NC-Task 1 SAF/Axes/Axis 8 PF1K0-WFS-MMS-Y
//     PlcTask Inputs/Main.M8.Axis.NcToPlc <-> Outputs/ToPlc
//     PlcTask Outputs/Main.M8.Axis.PlcToNc <-> Inputs/FromPlc
//   kfe_motion Instance <-> NC-Task 1 SAF/Axes/Axis 9 PF1K0-WFS-MMS-Z
//     PlcTask Inputs/Main.M9.Axis.NcToPlc <-> Outputs/ToPlc
//     PlcTask Outputs/Main.M9.Axis.PlcToNc <-> Inputs/FromPlc
//   kfe_motion Instance <-> NC-Task 1 SAF/Axes/SL1K0-BOTTOM-M21
//     PlcTask Inputs/Main.M21.Axis.NcToPlc <-> Outputs/ToPlc
//     PlcTask Outputs/Main.M21.Axis.PlcToNc <-> Inputs/FromPlc
//   kfe_motion Instance <-> NC-Task 1 SAF/Axes/SL1K0-NORTH-M20
//     PlcTask Inputs/Main.M20.Axis.NcToPlc <-> Outputs/ToPlc
//     PlcTask Outputs/Main.M20.Axis.PlcToNc <-> Inputs/FromPlc
//   kfe_motion Instance <-> NC-Task 1 SAF/Axes/SL1K0-SOUTH-M18
//     PlcTask Inputs/Main.M18.Axis.NcToPlc <-> Outputs/ToPlc
//     PlcTask Outputs/Main.M18.Axis.PlcToNc <-> Inputs/FromPlc
//   kfe_motion Instance <-> NC-Task 1 SAF/Axes/SL1K0-TOP-M19
//     PlcTask Inputs/Main.M19.Axis.NcToPlc <-> Outputs/ToPlc
//     PlcTask Outputs/Main.M19.Axis.PlcToNc <-> Inputs/FromPlc
//   kfe_motion Instance <-> NC-Task 1 SAF/Axes/SL2K0-BOTTOM-M25
//     PlcTask Inputs/Main.M25.Axis.NcToPlc <-> Outputs/ToPlc
//     PlcTask Outputs/Main.M25.Axis.PlcToNc <-> Inputs/FromPlc
//   kfe_motion Instance <-> NC-Task 1 SAF/Axes/SL2K0-NORTH-M24
//     PlcTask Inputs/Main.M24.Axis.NcToPlc <-> Outputs/ToPlc
//     PlcTask Outputs/Main.M24.Axis.PlcToNc <-> Inputs/FromPlc
//   kfe_motion Instance <-> NC-Task 1 SAF/Axes/SL2K0-SOUTH-M22
//     PlcTask Inputs/Main.M22.Axis.NcToPlc <-> Outputs/ToPlc
//     PlcTask Outputs/Main.M22.Axis.PlcToNc <-> Inputs/FromPlc
//   kfe_motion Instance <-> NC-Task 1 SAF/Axes/SL2K0-TOP-M23
//     PlcTask Inputs/Main.M23.Axis.NcToPlc <-> Outputs/ToPlc
//     PlcTask Outputs/Main.M23.Axis.PlcToNc <-> Inputs/FromPlc
//   kfe_motion Instance <-> NC-Task 1 SAF/Axes/ST1K4-TEST
//     PlcTask Inputs/Main.M33.Axis.NcToPlc <-> Outputs/ToPlc
//     PlcTask Outputs/Main.M33.Axis.PlcToNc <-> Inputs/FromPlc

CONFIGURATION kfe_motion
    RESOURCE PLC ON TwinCAT3
        TASK PlcTask(INTERVAL := T#10ms, PRIORITY := 20);
        PROGRAM PRG_1_PlcTask WITH PlcTask : PRG_1_PlcTask;
    END_RESOURCE
END_CONFIGURATION

// ---- GVLs/Main.TcGVL
{attribute 'qualified_only'}
VAR_GLOBAL
(*
    Only includes motor definitions for the IOC
    These are hard-coded to be Main.M#,
    but are very convenient to store in a GVL,
    hence the confusing namespace here

    This should be refactored once the IOC
    supports arbitrary ads paths for motors
*)
    // IM1K0-XTES: 3 Axes
    {attribute 'pytmc' := 'pv: IM1K0:XTES:MMS'}
    {attribute 'TcLinkTo' := '.bLimitForwardEnable  := TIIB[IM1K0-EL7041]^STM Status^Status^Digital input 1;
                              .bBrakeRelease        := TIIB[IM1K0-EL2004]^Channel 1^Output;
                              .nRawEncoderINT       := TIIB[IM1K0-EL3054]^AI Standard Channel 1^Value'}
    M1: ST_MotionStage := (sName := 'IM1K0:XTES:MMS');
    {attribute 'pytmc' := 'pv: IM1K0:XTES:CLZ'}
    {attribute 'TcLinkTo' := '.bHome                := TIIB[IM1K0-EL1088]^Channel 2^Input;
                              .nRawEncoderUINT      := TIIB[IM1K0-EL5101-01]^ENC Status compact^Counter value'}
    M2: ST_MotionStage := (sName := 'IM1K0:XTES:CLZ');
    {attribute 'pytmc' := 'pv: IM1K0:XTES:CLF'}
    {attribute 'TcLinkTo' := '.bHome                := TIIB[IM1K0-EL1088]^Channel 4^Input;
                              .nRawEncoderUINT      := TIIB[IM1K0-EL5101-01]^ENC Status compact^Counter value'}
    M3: ST_MotionStage := (sName := 'IM1K0:XTES:CLF');

    // IM1K3-PPM: 1 Axis
    {attribute 'pytmc' := 'pv: IM1K3:PPM:MMS'}
    {attribute 'TcLinkTo' := '.bLimitForwardEnable  := TIIB[IM1K3-EL7041]^STM Status^Status^Digital input 1;
                              .bLimitBackwardEnable := TIIB[IM1K3-EL7041]^STM Status^Status^Digital input 2;
                              .bBrakeRelease        := TIIB[IM1K3-EL2004]^Channel 1^Output;
                              .nRawEncoderULINT     := TIIB[IM1K3-EL5042]^FB Inputs Channel 1^Position'}
    M4: ST_MotionStage := (sName := 'IM1K3:PPM:MMS');
	
    // IM2K0-XTES: 1 Axis, previously 3 but the zoom/focus have been removed
    {attribute 'pytmc' := 'pv: IM2K0:XTES:MMS'}
    {attribute 'TcLinkTo' := '.bBrakeRelease        := TIIB[IM2K0-EL2004]^Channel 1^Output;
                              .nRawEncoderULINT     := TIIB[IM2K0-EL5042]^FB Inputs Channel 1^Position'}
    M5: ST_MotionStage := (sName := 'IM2K0:XTES:MMS');
    {attribute 'pytmc' := 'pv: IM2K0:XTES:CLZ'}
    {attribute 'TcLinkTo' := '.bHome                := TIIB[IM2K0-EL1088]^Channel 2^Input;
                              .nRawEncoderUINT      := TIIB[IM2K0-EL7342]^ENC Status compact Channel 1^Counter value'}
    M6: ST_MotionStage := (sName := 'IM2K0:XTES:CLZ');
    {attribute 'pytmc' := 'pv: IM2K0:XTES:CLF'}
    {attribute 'TcLinkTo' := '.bHome                := TIIB[IM2K0-EL1088]^Channel 4^Input;
                              .nRawEncoderUINT      := TIIB[IM2K0-EL7342]^ENC Status compact Channel 2^Counter value'}
    M7: ST_MotionStage := (sName := 'IM2K0:XTES:CLF');

    // PF1K0-WFS: 2 Axes
    {attribute 'pytmc' := 'pv: PF1K0:WFS:MMS:Y'}
    {attribute 'TcLinkTo' := '.bLimitForwardEnable  := TIIB[PF1K0-EL7041-01]^STM Status^Status^Digital input 1;
                              .bLimitBackwardEnable := TIIB[PF1K0-EL7041-01]^STM Status^Status^Digital input 2;
                              .bBrakeRelease        := TIIB[PF1K0-EL2004]^Channel 1^Output;
                              .nRawEncoderULINT     := TIIB[PF1K0-EL5042]^FB Inputs Channel 2^Position'}
    M8: ST_MotionStage := (sName := 'PF1K0:WFS:MMS:Y');
    {attribute 'pytmc' := 'pv: PF1K0:WFS:MMS:Z'}
    {attribute 'TcLinkTo' := '.nRawEncoderULINT     := TIIB[PF1K0-EL5042]^FB Inputs Channel 1^Position'}
    M9: ST_MotionStage := (sName := 'PF1K0:WFS:MMS:Z');

   // RTDSK0: 8 Axes
    M10: ST_MotionStage;
    {attribute 'pytmc' := 'pv: RTDSK0:SCRP:MMS:Z'}
    {attribute 'TcLinkTo' := '.bLimitForwardEnable  := TIIB[RTDSK0-M2-EL7041]^STM Status^Status^Digital input 1;
                              .bLimitBackwardEnable := TIIB[RTDSK0-M2-EL7041]^STM Status^Status^Digital input 2'}
    M11: ST_MotionStage:= (sName := 'RTDSK0:SCRP:MMS:Z');
        {attribute 'pytmc' := 'pv: RTDSK0:SCRP:MMS:X'}
    {attribute 'TcLinkTo' := '.bLimitForwardEnable  := TIIB[RTDSK0-M3-EL7041]^STM Status^Status^Digital input 1;
                              .bLimitBackwardEnable := TIIB[RTDSK0-M3-EL7041]^STM Status^Status^Digital input 2'}
    M12: ST_MotionStage:= (sName := 'RTDSK0:SCRP:MMS:X');
        {attribute 'pytmc' := 'pv: RTDSK0:SCRP:MMS:Y'}
    {attribute 'TcLinkTo' := '.bLimitForwardEnable  := TIIB[RTDSK0-M4-EL7041]^STM Status^Status^Digital input 1;
                              .bLimitBackwardEnable := TIIB[RTDSK0-M4-EL7041]^STM Status^Status^Digital input 2'}
    M13: ST_MotionStage:= (sName := 'RTDSK0:SCRP:MMS:Y');
    M14: ST_MotionStage;
    M15: ST_MotionStage;
    M16: ST_MotionStage;
    M17: ST_MotionStage;

    // SL1K0-POWER: 4 Axes
    {attribute 'pytmc' := 'pv: SL1K0:POWER:MMS:SOUTH'}
    {attribute 'TcLinkTo' := '.bLimitForwardEnable  := TIIB[SL1K0-EL7041-E1]^STM Status^Status^Digital input 2;
                              .bLimitBackwardEnable := TIIB[SL1K0-EL7041-E1]^STM Status^Status^Digital input 1;
                              .nRawEncoderINT       := TIIB[SL1K0-EL3054-E12]^AI Standard Channel 1^Value'}

    M18: ST_MotionStage := (sName := 'SL1K0:POWER:MMS:SOUTH');
    {attribute 'pytmc' := 'pv: SL1K0:POWER:MMS:TOP'}
    {attribute 'TcLinkTo' := '.bLimitForwardEnable  := TIIB[SL1K0-EL7041-E2]^STM Status^Status^Digital input 2;
                              .bLimitBackwardEnable := TIIB[SL1K0-EL7041-E2]^STM Status^Status^Digital input 1;
                              .nRawEncoderINT       := TIIB[SL1K0-EL3054-E12]^AI Standard Channel 2^Value'}
    M19: ST_MotionStage := (sName := 'SL1K0:POWER:MMS:TOP');
    {attribute 'pytmc' := 'pv: SL1K0:POWER:MMS:NORTH'}
    {attribute 'TcLinkTo' := '.bLimitForwardEnable  := TIIB[SL1K0-EL7041-E4]^STM Status^Status^Digital input 2;
                              .bLimitBackwardEnable := TIIB[SL1K0-EL7041-E4]^STM Status^Status^Digital input 1;
                              .nRawEncoderINT       := TIIB[SL1K0-EL3054-E12]^AI Standard Channel 3^Value'}
    M20: ST_MotionStage := (sName := 'SL1K0:POWER:MMS:NORTH');
    {attribute 'pytmc' := 'pv: SL1K0:POWER:MMS:BOTTOM'}
    {attribute 'TcLinkTo' := '.bLimitForwardEnable  := TIIB[SL1K0-EL7041-E5]^STM Status^Status^Digital input 2;
                              .bLimitBackwardEnable := TIIB[SL1K0-EL7041-E5]^STM Status^Status^Digital input 1;
                              .nRawEncoderINT       := TIIB[SL1K0-EL3054-E12]^AI Standard Channel 4^Value'}
    M21: ST_MotionStage := (sName := 'SL1K0:POWER:MMS:BOTTOM');

    // SL2K0-POWER: 4 Axes
    {attribute 'pytmc' := 'pv: SL2K0:POWER:MMS:SOUTH'}
    {attribute 'TcLinkTo' := '.bLimitForwardEnable  := TIIB[SL2K0-EL7041-E1]^STM Status^Status^Digital input 2;
                              .bLimitBackwardEnable := TIIB[SL2K0-EL7041-E1]^STM Status^Status^Digital input 1;
                              .nRawEncoderUINT      := TIIB[SL2K0-EL5042-E2]^FB Inputs Channel 1^Position'}
    M22: ST_MotionStage := (sName := 'SL2K0:POWER:MMS:SOUTH');
    {attribute 'pytmc' := 'pv: SL2K0:POWER:MMS:TOP'}
    {attribute 'TcLinkTo' := '.bLimitForwardEnable  := TIIB[SL2K0-EL7041-E3]^STM Status^Status^Digital input 2;
                              .bLimitBackwardEnable := TIIB[SL2K0-EL7041-E3]^STM Status^Status^Digital input 1;
                              .nRawEncoderUINT      := TIIB[SL2K0-EL5042-E2]^FB Inputs Channel 2^Position'}
    M23: ST_MotionStage := (sName := 'SL2K0:POWER:MMS:TOP');
    {attribute 'pytmc' := 'pv: SL2K0:POWER:MMS:NORTH'}
    {attribute 'TcLinkTo' := '.bLimitForwardEnable  := TIIB[SL2K0-EL7041-E5]^STM Status^Status^Digital input 2;
                              .bLimitBackwardEnable := TIIB[SL2K0-EL7041-E5]^STM Status^Status^Digital input 1;
                              .nRawEncoderUINT      := TIIB[SL2K0-EL5042-E6]^FB Inputs Channel 1^Position'}
    M24: ST_MotionStage := (sName := 'SL2K0:POWER:MMS:NORTH');
    {attribute 'pytmc' := 'pv: SL2K0:POWER:MMS:BOTTOM'}
    {attribute 'TcLinkTo' := '.bLimitForwardEnable  := TIIB[SL2K0-EL7041-E7]^STM Status^Status^Digital input 2;
                              .bLimitBackwardEnable := TIIB[SL2K0-EL7041-E7]^STM Status^Status^Digital input 1;
                              .nRawEncoderUINT      := TIIB[SL2K0-EL5042-E6]^FB Inputs Channel 2^Position'}
    M25: ST_MotionStage := (sName := 'SL2K0:POWER:MMS:BOTTOM');

    // AT1K4-SOLID: 4 axes (Z=748)
    (* Important note

        AT1K4 axes were mistakenly wired opposite to other solid attenuators.
        The intended convention is:
            MMS:01 should be the most upstream blade,
            MMS:04 should be the most downstream blade.

        The fix applied here is that the NC axes and temperature sensors are *linked* in reverse.
        In summary:

        Traveler	EPICS	Stage		NC	Location
        Axis 4		MMS:01	fbStage1	26	Upstream
        Axis 3		MMS:02	fbStage2	27
        Axis 2		MMS:03	fbStage3	28
        Axis 1		MMS:04	fbStage4	29	Downstream

    *)
    {attribute 'pytmc' := 'pv: AT1K4:L2SI:MMS:01'}
    {attribute 'TcLinkTo' := '
        .bLimitForwardEnable  := TIIB[AT1K4-EL7047-04]^STM Status^Status^Digital input 1;
        .bLimitBackwardEnable := TIIB[AT1K4-EL7047-04]^STM Status^Status^Digital input 2;
        .nRawEncoderULINT     := TIIB[AT1K4-EL5042-02]^FB Inputs Channel 2^Position;
    '}
    M26: ST_MotionStage := (sName := 'AT1K4:L2SI:MMS:01');

    {attribute 'pytmc' := 'pv: AT1K4:L2SI:MMS:02'}
    {attribute 'TcLinkTo' := '
        .bLimitForwardEnable  := TIIB[AT1K4-EL7047-03]^STM Status^Status^Digital input 1;
        .bLimitBackwardEnable := TIIB[AT1K4-EL7047-03]^STM Status^Status^Digital input 2;
        .nRawEncoderULINT     := TIIB[AT1K4-EL5042-02]^FB Inputs Channel 1^Position;
    '}
    M27: ST_MotionStage := (sName := 'AT1K4:L2SI:MMS:02');

    {attribute 'pytmc' := 'pv: AT1K4:L2SI:MMS:03'}
    {attribute 'TcLinkTo' := '
        .bLimitForwardEnable  := TIIB[AT1K4-EL7047-02]^STM Status^Status^Digital input 1;
        .bLimitBackwardEnable := TIIB[AT1K4-EL7047-02]^STM Status^Status^Digital input 2;
        .nRawEncoderULINT     := TIIB[AT1K4-EL5042-01]^FB Inputs Channel 2^Position;
    '}
    M28: ST_MotionStage := (sName := 'AT1K4:L2SI:MMS:03');

    {attribute 'pytmc' := 'pv: AT1K4:L2SI:MMS:04'}
    {attribute 'TcLinkTo' := '
        .bLimitForwardEnable  := TIIB[AT1K4-EL7047-01]^STM Status^Status^Digital input 1;
        .bLimitBackwardEnable := TIIB[AT1K4-EL7047-01]^STM Status^Status^Digital input 2;
        .nRawEncoderULINT     := TIIB[AT1K4-EL5042-01]^FB Inputs Channel 1^Position;
    '}
    M29: ST_MotionStage := (sName := 'AT1K4:L2SI:MMS:04');

    // IM1K4-XTES: 3 Axes
    {attribute 'pytmc' := 'pv: IM1K4:XTES:MMS'}
    {attribute 'TcLinkTo' := '.bLimitForwardEnable  := TIIB[IM1K4-EL7041-E1]^STM Status^Status^Digital input 1;
                              .bBrakeRelease        := TIIB[IM1K4-EL2004-E2]^Channel 1^Output;
                              .nRawEncoderULINT     := TIIB[IM1K4-EL5042-E3]^FB Inputs Channel 1^Position'}
    M30: ST_MotionStage := (sName := 'IM1K4:XTES:MMS');
    {attribute 'pytmc' := 'pv: IM1K4:XTES:CLZ'}
    {attribute 'TcLinkTo' := '.bHome                := TIIB[IM1K4-EL1088-E5]^Channel 2^Input;
                              .nRawEncoderUINT     := TIIB[IM1K4-EL7342-E4]^ENC Status compact Channel 1^Counter value'}
    M31: ST_MotionStage := (sName := 'IM1K4:XTES:CLZ');
    {attribute 'pytmc' := 'pv: IM1K4:XTES:CLF'}
    {attribute 'TcLinkTo' := '.bHome := TIIB[IM1K4-EL1088-E5]^Channel 4^Input;
                              .nRawEncoderUINT     := TIIB[IM1K4-EL7342-E4]^ENC Status compact Channel 2^Counter value'}
    M32: ST_MotionStage := (sName := 'IM1K4:XTES:CLF');

    // ST1K4-TEST: 1 Axis
    {attribute 'pytmc' := 'pv: ST1K4:TEST:MMS:01'}
    {attribute 'TcLinkTo' := '.bLimitForwardEnable  := TIIB[ST1K4-EL7041-E4]^STM Status^Status^Digital input 1;
                              .bLimitBackwardEnable := TIIB[ST1K4-EL7041-E4]^STM Status^Status^Digital input 2;
                              .bBrakeRelease        := TIIB[ST1K4-EL2202-E3]^Channel 1^Output;
                              .nRawEncoderULINT      := TIIB[ST1K4-EL5042-E6]^FB Inputs Channel 1^Position'}
    M33: ST_MotionStage := (sName := 'ST1K4:TEST:MMS:01');
END_VAR

// ---- GVLs/GVL.TcGVL
{attribute 'qualified_only'}
VAR_GLOBAL
    {attribute 'pytmc' := 'pv: PLC:KFE:MOTION:ARB:01'}
    fbArbiter: FB_Arbiter(1);
    {attribute 'pytmc' := 'pv: PLC:KFE:MOTION:ARB:02'}
    fbArbiter2: FB_Arbiter(2);
    {attribute 'pytmc' := 'pv: PLC:KFE:MOTION:ARB:03'}
    fbArbiter3: FB_Arbiter(3);
    {attribute 'pytmc' := 'pv: PLC:KFE:MOTION:FFO:01'}
    {attribute 'TcLinkTo' := '.q_xFastFaultOut:=TIIB[PMPS_FFO]^Channel 1^Output'}
    fbFastFaultOutput1: FB_HardwareFFOutput := (bAutoReset := TRUE, i_sNetID:='172.21.92.73.1.1');
    {attribute 'pytmc' := 'pv: PLC:KFE:MOTION:FFO:02'}
    {attribute 'TcLinkTo' := '.q_xFastFaultOut:=TIIB[PMPS_FFO]^Channel 2^Output'}
    fbFastFaultOutput2: FB_HardwareFFOutput := (bAutoReset := TRUE, i_sNetID:='172.21.92.73.1.1');
    {attribute 'pytmc' := 'pv: PLC:KFE:MOTION:FFO:03'}
    fbFastFaultOutput3: FB_HardwareFFOutput := (bAutoReset := TRUE, i_sNetID:='172.21.92.73.1.1');

    {attribute 'pytmc' := 'pv: PLC:KFE:MOTION:PMPS:ReqTrans'}
    rReqTrans AT %I*		: ARRAY [1..PMPS_GVL.AUX_ATTENUATORS] OF ST_PMPS_Attenuator_IO;
    {attribute 'pytmc' := 'pv: PLC:KFE:MOTION:PMPS:CurTrans'}
    rCurTrans AT %Q*		: ARRAY [1..PMPS_GVL.AUX_ATTENUATORS] OF ST_PMPS_Attenuator_IO;

    ePF1K0State: E_WFS_States;

     {attribute 'TcLinkTo' := 'TIIB[PMPS_PRE]^IO Outputs^ST1K4_Y_ENC'}
    PMPS_ST1K4_Y_ENC AT%Q* : UDINT;
END_VAR

VAR_GLOBAL CONSTANT
    iFiltersPerSATTBlade : INT := 8;
END_VAR

// ---- POUs/PRG_1_PlcTask.TcPOU
PROGRAM PRG_1_PlcTask
VAR
END_VAR

PRG_2_PMPS_PRE();

PRG_IM1K0_XTES();
PRG_IM1K3_PPM();
PRG_IM2K0_XTES();
PRG_PF1K0_WFS();
PRG_PF1K0_PM();
PRG_RTDSK0();
PRG_SL1K0_POWER();
PRG_SL2K0_POWER();

PRG_AT1K4_SOLID();
PRG_IM1K4_XTES();
PRG_ST1K4_TEST();
PRG_OTHER();

PRG_3_PMPS_POST();
PRG_4_LOG();

END_PROGRAM

// ---- POUs/PRG_2_PMPS_PRE.TcPOU
PROGRAM PRG_2_PMPS_PRE
VAR
END_VAR

MOTION_GVL.fbStandardPMPSDB(
    io_fbFFHWO:=GVL.fbFastFaultOutput1,
    bEnable:=TRUE,
    sPLCName:='plc-kfe-motion',
);

END_PROGRAM

// ---- POUs/PRG_IM1K0_XTES.TcPOU
PROGRAM PRG_IM1K0_XTES
VAR
    {attribute 'pytmc' := 'pv: IM1K0:XTES'}
    {attribute 'TcLinkTo' := '.bZoomEndFwd := TIIB[IM1K0-EL1088]^Channel 1^Input;
                              .bZoomEndBwd := TIIB[IM1K0-EL1088]^Channel 2^Input;
                              .bFocusEndFwd := TIIB[IM1K0-EL1088]^Channel 3^Input;
                              .bFocusEndBwd := TIIB[IM1K0-EL1088]^Channel 4^Input;
                              .fbOpal.bOpalPower := TIIB[IM1K0-EL2004]^Channel 2^Output;
                              .fbLED.bLedPower := TIIB[IM1K0-EL2004]^Channel 3^Output;
                              .fbFlowSwitch.bFlowOk := TIIB[IM1K0-EL1004]^Channel 2^Input
'}
    fbIM1K0: FB_XPIM;
    fbStateSetup: FB_StateSetupHelper;
    stDefault: ST_PositionState := (
        fVelocity := 1,
        bMoveOk := TRUE,
        bValid := TRUE
    );
    {attribute 'TcLinkTo' := '.Status := TIIB[IM1K0-EL6002]^COM TxPDO-Map Inputs Channel 1^Status;
                              .D[0] := TIIB[IM1K0-EL6002]^COM TxPDO-Map Inputs Channel 1^Data In 0;
                              .D[1] := TIIB[IM1K0-EL6002]^COM TxPDO-Map Inputs Channel 1^Data In 1;
                              .D[2] := TIIB[IM1K0-EL6002]^COM TxPDO-Map Inputs Channel 1^Data In 2;
                              .D[3] := TIIB[IM1K0-EL6002]^COM TxPDO-Map Inputs Channel 1^Data In 3;
                              .D[4] := TIIB[IM1K0-EL6002]^COM TxPDO-Map Inputs Channel 1^Data In 4;
                              .D[5] := TIIB[IM1K0-EL6002]^COM TxPDO-Map Inputs Channel 1^Data In 5;
                              .D[6] := TIIB[IM1K0-EL6002]^COM TxPDO-Map Inputs Channel 1^Data In 6;
                              .D[7] := TIIB[IM1K0-EL6002]^COM TxPDO-Map Inputs Channel 1^Data In 7;
                              .D[8] := TIIB[IM1K0-EL6002]^COM TxPDO-Map Inputs Channel 1^Data In 8;
                              .D[9] := TIIB[IM1K0-EL6002]^COM TxPDO-Map Inputs Channel 1^Data In 9;
                              .D[10] := TIIB[IM1K0-EL6002]^COM TxPDO-Map Inputs Channel 1^Data In 10;
                              .D[11] := TIIB[IM1K0-EL6002]^COM TxPDO-Map Inputs Channel 1^Data In 11;
                              .D[12] := TIIB[IM1K0-EL6002]^COM TxPDO-Map Inputs Channel 1^Data In 12;
                              .D[13] := TIIB[IM1K0-EL6002]^COM TxPDO-Map Inputs Channel 1^Data In 13;
                              .D[14] := TIIB[IM1K0-EL6002]^COM TxPDO-Map Inputs Channel 1^Data In 14;
                              .D[15] := TIIB[IM1K0-EL6002]^COM TxPDO-Map Inputs Channel 1^Data In 15;
                              .D[16] := TIIB[IM1K0-EL6002]^COM TxPDO-Map Inputs Channel 1^Data In 16;
                              .D[17] := TIIB[IM1K0-EL6002]^COM TxPDO-Map Inputs Channel 1^Data In 17;
                              .D[18] := TIIB[IM1K0-EL6002]^COM TxPDO-Map Inputs Channel 1^Data In 18;
                              .D[19] := TIIB[IM1K0-EL6002]^COM TxPDO-Map Inputs Channel 1^Data In 19;
                              .D[20] := TIIB[IM1K0-EL6002]^COM TxPDO-Map Inputs Channel 1^Data In 20;
                              .D[21] := TIIB[IM1K0-EL6002]^COM TxPDO-Map Inputs Channel 1^Data In 21'}
    stEL6In AT %I*: EL6InData22b;
    {attribute 'TcLinkTo' := '.Ctrl := TIIB[IM1K0-EL6002]^COM RxPDO-Map Outputs Channel 1^Ctrl;
                              .D[0] := TIIB[IM1K0-EL6002]^COM RxPDO-Map Outputs Channel 1^Data Out 0;
                              .D[1] := TIIB[IM1K0-EL6002]^COM RxPDO-Map Outputs Channel 1^Data Out 1;
                              .D[2] := TIIB[IM1K0-EL6002]^COM RxPDO-Map Outputs Channel 1^Data Out 2;
                              .D[3] := TIIB[IM1K0-EL6002]^COM RxPDO-Map Outputs Channel 1^Data Out 3;
                              .D[4] := TIIB[IM1K0-EL6002]^COM RxPDO-Map Outputs Channel 1^Data Out 4;
                              .D[5] := TIIB[IM1K0-EL6002]^COM RxPDO-Map Outputs Channel 1^Data Out 5;
                              .D[6] := TIIB[IM1K0-EL6002]^COM RxPDO-Map Outputs Channel 1^Data Out 6;
                              .D[7] := TIIB[IM1K0-EL6002]^COM RxPDO-Map Outputs Channel 1^Data Out 7;
                              .D[8] := TIIB[IM1K0-EL6002]^COM RxPDO-Map Outputs Channel 1^Data Out 8;
                              .D[9] := TIIB[IM1K0-EL6002]^COM RxPDO-Map Outputs Channel 1^Data Out 9;
                              .D[10] := TIIB[IM1K0-EL6002]^COM RxPDO-Map Outputs Channel 1^Data Out 10;
                              .D[11] := TIIB[IM1K0-EL6002]^COM RxPDO-Map Outputs Channel 1^Data Out 11;
                              .D[12] := TIIB[IM1K0-EL6002]^COM RxPDO-Map Outputs Channel 1^Data Out 12;
                              .D[13] := TIIB[IM1K0-EL6002]^COM RxPDO-Map Outputs Channel 1^Data Out 13;
                              .D[14] := TIIB[IM1K0-EL6002]^COM RxPDO-Map Outputs Channel 1^Data Out 14;
                              .D[15] := TIIB[IM1K0-EL6002]^COM RxPDO-Map Outputs Channel 1^Data Out 15;
                              .D[16] := TIIB[IM1K0-EL6002]^COM RxPDO-Map Outputs Channel 1^Data Out 16;
                              .D[17] := TIIB[IM1K0-EL6002]^COM RxPDO-Map Outputs Channel 1^Data Out 17;
                              .D[18] := TIIB[IM1K0-EL6002]^COM RxPDO-Map Outputs Channel 1^Data Out 18;
                              .D[19] := TIIB[IM1K0-EL6002]^COM RxPDO-Map Outputs Channel 1^Data Out 19;
                              .D[20] := TIIB[IM1K0-EL6002]^COM RxPDO-Map Outputs Channel 1^Data Out 20;
                              .D[21] := TIIB[IM1K0-EL6002]^COM RxPDO-Map Outputs Channel 1^Data Out 21'}
    stEL6Out AT %Q*: EL6OutData22b;
END_VAR


fbStateSetup(stPositionState:=stDefault, bSetDefault:=TRUE);

fbStateSetup(stPositionState:=fbIM1K0.stOut, fPosition:=0, sPmpsState:='IM1K0:XTES-OUT');
fbStateSetup(stPositionState:=fbIM1K0.stYag, fPosition:=-27.65, sPmpsState:='IM1K0:XTES-YAG');
fbStateSetup(stPositionState:=fbIM1K0.stDiamond, fPosition:=-57.65, sPmpsState:='IM1K0:XTES-DIAMOND');
fbStateSetup(stPositionState:=fbIM1K0.stReticle, fPosition:=-87.65, sPmpsState:='IM1K0:XTES-RETICLE');

fbIM1K0(
    fbFFHWO := GVL.fbFastFaultOutput1,
    fbArbiter := GVL.fbArbiter,
    stYStage := Main.M1,
    stZoomStage := Main.M2,
    stFocusStage := Main.M3,
    stEl6In := stEL6In,
    stEl6Out := stEl6Out,
    sDeviceName := 'IM1K0:XTES',
    sTransitionKey := 'IM1K0:XTES-TRANSITION',
    bEnableMotion := TRUE,
    bEnableBeamParams := TRUE,
    bEnablePositionLimits := TRUE,
);

END_PROGRAM

// ---- POUs/PRG_IM1K3_PPM.TcPOU
PROGRAM PRG_IM1K3_PPM
VAR
    {attribute 'pytmc' := 'pv: IM1K3:PPM'}
    {attribute 'TcLinkTo' := '.fbGige.iIlluminatorINT := TIIB[IM1K3-EL4004]^AO Outputs Channel 1^Analog output;
                              .fbGige.bGigePower := TIIB[IM1K3-EL2004]^Channel 2^Output;
                              .fbPowerMeter.iVoltageINT := TIIB[IM1K3-EL3062]^AI Standard Channel 1^Value;
                              .fbPowerMeter.fbThermoCouple.bError := TIIB[IM1K3-EL3314]^TC Inputs Channel 1^Status^Error;
                              .fbPowerMeter.fbThermoCouple.bUnderrange := TIIB[IM1K3-EL3314]^TC Inputs Channel 1^Status^Underrange;
                              .fbPowerMeter.fbThermoCouple.bOverrange := TIIB[IM1K3-EL3314]^TC Inputs Channel 1^Status^Overrange;
                              .fbPowerMeter.fbThermoCouple.iRaw := TIIB[IM1K3-EL3314]^TC Inputs Channel 1^Value;
                              .fbYagThermoCouple.bError := TIIB[IM1K3-EL3314]^TC Inputs Channel 2^Status^Error;
                              .fbYagThermoCouple.bUnderrange := TIIB[IM1K3-EL3314]^TC Inputs Channel 2^Status^Underrange;
                              .fbYagThermoCouple.bOverrange := TIIB[IM1K3-EL3314]^TC Inputs Channel 2^Status^Overrange;
                              .fbYagThermoCouple.iRaw := TIIB[IM1K3-EL3314]^TC Inputs Channel 2^Value;
                              .fbFlowSwitch.bFlowOk := TIIB[ST1K4-EL1004-E5]^Channel 3^Input'}
    fbIM1K3: FB_PPM;
    fbStateSetup: FB_StateSetupHelper;
    stDefault: ST_PositionState := (
        fVelocity := 15,
        bMoveOk := TRUE,
        bValid := TRUE
    );

END_VAR


fbStateSetup(stPositionState:=stDefault, bSetDefault:=TRUE);

fbStateSetup(stPositionState:=fbIM1K3.stOut, fPosition:=-9.1, sPmpsState:='IM1K3:PPM-OUT');
fbStateSetup(stPositionState:=fbIM1K3.stPower, fPosition:=-48.2, sPmpsState:='IM1K3:PPM-POWERMETER');
fbStateSetup(stPositionState:=fbIM1K3.stYag1, fPosition:=-72.2, sPmpsState:='IM1K3:PPM-YAG1');
fbStateSetup(stPositionState:=fbIM1K3.stYag2, fPosition:=-98.21, sPmpsState:='IM1K3:PPM-YAG2');

fbIM1K3(
    fbFFHWO := GVL.fbFastFaultOutput3,
    fbArbiter := GVL.fbArbiter3,
    stYStage := Main.M4,
    sDeviceName := 'IM1K3:PPM',
    sTransitionKey := 'IM1K3:PPM-TRANSITION',
    bEnableMotion := TRUE,
    bEnableBeamParams := TRUE,
    bEnablePositionLimits := TRUE,
);

END_PROGRAM

// ---- POUs/PRG_IM2K0_XTES.TcPOU
PROGRAM PRG_IM2K0_XTES
VAR
    {attribute 'pytmc' := 'pv: IM2K0:XTES'}
    {attribute 'TcLinkTo' := '.fbLED.bLedPower := TIIB[IM2K0-EL2004]^Channel 3^Output;
                              .fbGige.bGigePower := TIIB[IM2K0-EL2004]^Channel 4^Output;
                              .fbFlowSwitch.bFlowOk := TIIB[SL2K0-EL1004-E12]^Channel 1^Input'} // same cooling loop as SL2K0
    fbIM2K0: FB_XPIM_IM2K0;
    fbStateSetup: FB_StateSetupHelper;
    stDefault: ST_PositionState := (
        fVelocity := 1,
        bMoveOk := TRUE,
        bValid := TRUE
    );

    {attribute 'TcLinkTo' := 'TIIB[IM2K0-EL7041]^STM Status^Status^Digital input 1'}
    bDefectiveLimitSwitch AT %I*: BOOL;
END_VAR


fbStateSetup(stPositionState:=stDefault, bSetDefault:=TRUE);

fbStateSetup(stPositionState:=fbIM2K0.stOut, fPosition:=0, sPmpsState:='IM2K0:XTES-OUT');
fbStateSetup(stPositionState:=fbIM2K0.stYag, fPosition:=-87.65);
fbStateSetup(stPositionState:=fbIM2K0.stDiamond, fPosition:=-57.65, sPmpsState:='IM2K0:XTES-DIAMOND');
fbStateSetup(stPositionState:=fbIM2K0.stReticle, fPosition:=-27.65, sPmpsState:='IM2K0:XTES-RETICLE');

CASE GVL.ePF1K0State OF
    E_WFS_STATES.TARGET1, E_WFS_STATES.TARGET2, E_WFS_STATES.TARGET3, E_WFS_STATES.TARGET4, E_WFS_STATES.TARGET5 :
        // Known state targets: allow less strict pmps
        fbIM2K0.stYag.stPMPS.sPmpsState := 'IM2K0:XTES-YAG_WFS_IN';
ELSE
    // Out, Unknown, or an unexpected state: full pmps
    fbIM2K0.stYag.stPMPS.sPmpsState := 'IM2K0:XTES-YAG';
END_CASE

fbIM2K0(
    fbFFHWO := GVL.fbFastFaultOutput1,
    fbArbiter := GVL.fbArbiter,
    stYStage := Main.M5,
    sDeviceName := 'IM2K0:XTES',
    sTransitionKey := 'IM2K0:XTES-TRANSITION',
    bEnableMotion := TRUE,
    bEnableBeamParams := TRUE,
    bEnablePositionLimits := TRUE,
);

Main.M5.bLimitForwardEnable := bDefectiveLimitSwitch OR (Main.M5.stAxisStatus.fActPosition < 0);

END_PROGRAM

// ---- POUs/IM2K0/FB_XPIM_IM2K0.TcPOU
FUNCTION_BLOCK FB_XPIM_IM2K0
(*
    Function block for the IM2K0 imager. This used to be a standard XPIM, but
    IM2K0 has been modified to replace the lens, illuminator, and camera with the PPM versions.

    This function block therefore controls:
    - Y motion (XPIM style)
    - Y scintillator states (XPIM style)
    - camera power (PPM style)
    - camera illuminator (PPM style but with XPIM style on/off only)
    - flowswitch (XPIM style, not fully implemented)
*)
VAR_IN_OUT
    // Y motor (state select).
    stYStage: ST_MotionStage;
    // The fast fault output to fault to.
    fbFFHWO: FB_HardwareFFOutput;
    // The arbiter to request beam conditions from.
    fbArbiter: FB_Arbiter;
END_VAR
VAR_INPUT
    // Settings for the OUT state.
    stOut: ST_PositionState;
    // Settings for the YAG state.
    stYag: ST_PositionState;
    // Settings for the DIAMOND state.
    stDiamond: ST_PositionState;
    // Settings for the RETICLE state.
    stReticle: ST_PositionState;
    // Set this to a non-unknown value to request a new move.
    {attribute 'pytmc' := '
        pv: MMS:STATE:SET
        io: io
    '}
    eEnumSet: E_XPIM_States;
    // Set this to TRUE to enable input state moves, or FALSE to disable them.
    bEnableMotion: BOOL;
    // Set this to TRUE to enable beam parameter checks, or FALSE to disable them.
    bEnableBeamParams: BOOL;
    // Set this to TRUE to enable position limit checks, or FALSE to disable them.
    bEnablePositionLimits: BOOL;
    // The name of the device for use in the PMPS DB lookup and diagnostic screens.
    sDeviceName: STRING;
    // The name of the transition state in the PMPS database.
    sTransitionKey: STRING;
    // Set this to TRUE to re-read the loaded database immediately (useful for debug).
    bReadDBNow: BOOL;
END_VAR
VAR_OUTPUT
    // The current position state as an enum.
    {attribute 'pytmc' := '
        pv: MMS:STATE:GET
        io: i
    '}
    eEnumGet: E_XPIM_States;
    // The PMPS database lookup associated with the current position state.
    stDbStateParams: ST_DbStateParams;
END_VAR
VAR
    bInit: BOOL;

    fbYStage: FB_MotionStage;

    fbStateDefaults: FB_PositionState_Defaults;

    {attribute 'pytmc' := '
        pv: MMS
        astPositionState.array: 1..4
    '}
    fbStates: FB_PositionStatePMPS1D;
    astPositionState: ARRAY[1..GeneralConstants.MAX_STATES] OF ST_PositionState;
    fbArrCheckWrite: FB_CheckPositionStateWrite;

    {attribute 'pytmc' := '
        pv: CAM
    '}
    fbGige: FB_PPM_Gige;

    {attribute 'pytmc' := '
        pv: CIL
    '}
    fbLED: FB_XPIM_LED;

    {attribute 'pytmc' := '
        pv: FSW
    '}
    fbFlowSwitch: FB_XTES_Flowswitch;
END_VAR
VAR CONSTANT
    // State defaults if not provided
    fDelta: LREAL := 2;
    fAccel: LREAL := 200;
    fOutDecel: LREAL := 25;
END_VAR


IF NOT bInit THEN
    bInit := TRUE;

    stYStage.bHardwareEnable := TRUE;
    stYStage.bPowerSelf := FALSE;
    // No limit switch at the bottom
    stYStage.bLimitBackwardEnable := TRUE;

    // Partial backcompat, this used to set fVelocity too but this should be set per install
    fbStateDefaults(stPositionState:=stOut, sNameDefault:='OUT', fDeltaDefault:=fDelta, fAccelDefault:=fAccel, fDecelDefault:=fOutDecel);
    fbStateDefaults(stPositionState:=stYag, sNameDefault:='YAG', fDeltaDefault:=fDelta, fAccelDefault:=fAccel, fDecelDefault:=fAccel);
    fbStateDefaults(stPositionState:=stDiamond, sNameDefault:='DIAMOND', fDeltaDefault:=fDelta, fAccelDefault:=fAccel, fDecelDefault:=fAccel);
    fbStateDefaults(stPositionState:=stReticle, sNameDefault:='RETICLE', fDeltaDefault:=fDelta, fAccelDefault:=fAccel, fDecelDefault:=fAccel);
END_IF

fbYStage(stMotionStage:=stYStage);

// We need to update from PLC or from EPICS, but not both
fbArrCheckWrite(
    astPositionState:=astPositionState,
    bCheck:=TRUE,
    bSave:=FALSE,
);
IF NOT fbArrCheckWrite.bHadWrite THEN
    astPositionState[E_XPIM_States.OUT] := stOut;
    astPositionState[E_XPIM_States.YAG] := stYag;
    astPositionState[E_XPIM_States.DIAMOND] := stDiamond;
    astPositionState[E_XPIM_States.RETICLE] := stReticle;
END_IF

fbStates(
    stMotionStage:=stYStage,
    astPositionState:=astPositionState,
    eEnumSet:=eEnumSet,
    eEnumGet:=eEnumGet,
    fbFFHWO:=fbFFHWO,
    fbArbiter:=fbArbiter,
    bEnableMotion:=bEnableMotion,
    bEnableBeamParams:=bEnableBeamParams,
    bEnablePositionLimits:=bEnablePositionLimits,
    sDeviceName:=sDeviceName,
    sTransitionKey:=sTransitionKey,
    bReadDBNow:=bReadDBNow,
    stDbStateParams=>stDbStateParams,
);

fbArrCheckWrite(
    astPositionState:=astPositionState,
    bCheck:=FALSE,
    bSave:=TRUE,
);

stOut := astPositionState[E_XPIM_States.OUT];
stYag := astPositionState[E_XPIM_States.YAG];
stDiamond := astPositionState[E_XPIM_States.DIAMOND];
stReticle := astPositionState[E_XPIM_States.RETICLE];

fbGige();
fbLED(enumXPIM:=eEnumGet);
fbFlowSwitch();

END_FUNCTION_BLOCK

// ---- POUs/PRG_PF1K0_WFS.TcPOU
PROGRAM PRG_PF1K0_WFS
VAR
    {attribute 'pytmc' := 'pv: PF1K0:WFS'}
    {attribute 'TcLinkTo' := '.fbThermoCouple1.bError := TIIB[PF1K0-EL3314]^TC Inputs Channel 1^Status^Error;
                              .fbThermoCouple1.bUnderrange := TIIB[PF1K0-EL3314]^TC Inputs Channel 1^Status^Underrange;
                              .fbThermoCouple1.bOverrange := TIIB[PF1K0-EL3314]^TC Inputs Channel 1^Status^Overrange;
                              .fbThermoCouple1.iRaw := TIIB[PF1K0-EL3314]^TC Inputs Channel 1^Value;
                              .fbThermoCouple2.bError := TIIB[PF1K0-EL3314]^TC Inputs Channel 2^Status^Error;
                              .fbThermoCouple2.bUnderrange := TIIB[PF1K0-EL3314]^TC Inputs Channel 2^Status^Underrange;
                              .fbThermoCouple2.bOverrange := TIIB[PF1K0-EL3314]^TC Inputs Channel 2^Status^Overrange;
                              .fbThermoCouple2.iRaw := TIIB[PF1K0-EL3314]^TC Inputs Channel 2^Value;
                              .fbFlowSwitch.bFlowOk := TIIB[SL2K0-EL1004-E12]^Channel 1^Input'} // shares same cooling loop as SL2K0
    fbPF1K0: FB_WFS;
    fbStateSetup: FB_StateSetupHelper;
    stDefault: ST_PositionState := (
        fVelocity := 1,
        bMoveOk := TRUE,
        bValid := TRUE
    );
END_VAR


fbStateSetup(stPositionState:=stDefault, bSetDefault:=TRUE);

fbStateSetup(stPositionState:=fbPF1K0.stOut, fPosition:=-15, sPmpsState:='PF1K0:WFS-OUT');
fbStateSetup(stPositionState:=fbPF1K0.stTarget1, fPosition:=-96.623, sPmpsState:='PF1K0:WFS-TARGET1');
fbStateSetup(stPositionState:=fbPF1K0.stTarget2, fPosition:=-82.25, sPmpsState:='PF1K0:WFS-TARGET2');
fbStateSetup(stPositionState:=fbPF1K0.stTarget3, fPosition:=-67.874, sPmpsState:='PF1K0:WFS-TARGET3');
fbStateSetup(stPositionState:=fbPF1K0.stTarget4, fPosition:=-53.5, sPmpsState:='PF1K0:WFS-TARGET4');
fbStateSetup(stPositionState:=fbPF1K0.stTarget5, fPosition:=-39.124, sPmpsState:='PF1K0:WFS-TARGET5');

fbPF1K0(
    fbFFHWO := GVL.fbFastFaultOutput1,
    fbArbiter := GVL.fbArbiter,
    stYStage := Main.M8,
    stZStage := Main.M9,
    sDeviceName := 'PF1K0:WFS',
    sTransitionKey := 'PF1K0:WFS-TRANSITION',
    bEnableMotion := TRUE,
    bEnableBeamParams := TRUE,
    bEnablePositionLimits := TRUE,
    eEnumGet => GVL.ePF1K0State,
);

END_PROGRAM

// ---- POUs/PRG_PF1K0_PM.TcPOU
PROGRAM PRG_PF1K0_PM
VAR
   {attribute 'TcLinkTo' := '.i_xInsertedLS := TIIB[PF1K0-MPA-EL1004]^Channel 1^Input;
                             .i_xRetractedLS := TIIB[PF1K0-MPA-EL1004]^Channel 2^Input;
                             .q_xInsert_DO :=  TIIB[PF1K0-MPA-EL2004]^Channel 1^Output;
                             .q_xRetract_DO :=  TIIB[PF1K0-MPA-EL2004]^Channel 2^Output
    '}

     {attribute 'pytmc' :=' pv: PF1K0:MPA:01 '}
    PF1K0_MPA_01: FB_MPA := (sName := 'PF1K0:PPM:MPA:01');

    {attribute 'pytmc' := 'pv: PF1K0:PM'}
    {attribute 'TcLinkTo' := '.iVoltageINT := TIIB[PF1K0-EL3062]^AI Standard Channel 1^Value;
                              .fbThermoCouple.bError := TIIB[PF1K0-EL3314]^TC Inputs Channel 1^Status^Error;
                              .fbThermoCouple.bUnderrange := TIIB[PF1K0-EL3314]^TC Inputs Channel 1^Status^Underrange;
                              .fbThermoCouple.bOverrange := TIIB[PF1K0-EL3314]^TC Inputs Channel 1^Status^Overrange;
                              .fbThermoCouple.iRaw := TIIB[PF1K0-EL3314]^TC Inputs Channel 1^Value;'}
    fbPowerMeter: FB_PPM_PowerMeter;
END_VAR


// Check Power Meter
fbPowerMeter();

// Act on MPA
PF1K0_MPA_01(
    ibInsertOK:= TRUE,
    ibRetractOK:= TRUE ,
    ibPMPS_OK:= TRUE ,
    ibOverrideInterlock:= ,
    q_stAct=> ,
    xMPS_OK=> ,
    xDone=> ,
    i_xReset := ,
    io_fbFFHWO := GVL.fbFastFaultOutput1,
);

END_PROGRAM

// ---- POUs/PRG_RTDSK0.TcPOU
PROGRAM PRG_RTDSK0
VAR

   {attribute 'TcLinkTo' := '.i_xInsertedLS := TIIB[RTDSK0-MPA-EL1008]^Channel 1^Input;
                             .i_xRetractedLS := TIIB[RTDSK0-MPA-EL1008]^Channel 2^Input;
                             .q_xInsert_DO :=  TIIB[RTDSK0-MPA-EL2008]^Channel 1^Output;
                             .q_xRetract_DO :=  TIIB[RTDSK0-MPA-EL2008]^Channel 2^Output
    '}

     {attribute 'pytmc' :=' pv: RTDSK0:MPA:01 '}
    RTDSK0_MPA_01: FB_MPA := (sName := 'RTDSK0:MPA:01');

   {attribute 'TcLinkTo' := '.i_xInsertedLS := TIIB[RTDSK0-MPA-EL1008]^Channel 3^Input;
                             .i_xRetractedLS := TIIB[RTDSK0-MPA-EL1008]^Channel 4^Input;
                             .q_xInsert_DO :=  TIIB[RTDSK0-MPA-EL2008]^Channel 3^Output;
                             .q_xRetract_DO :=  TIIB[RTDSK0-MPA-EL2008]^Channel 4^Output
    '}


    {attribute 'pytmc' :=' pv: RTDSK0:MPA:02 '}
    RTDSK0_MPA_02: FB_MPA := (sName := 'RTDSK0:MPA:02');

       {attribute 'TcLinkTo' := '.i_xInsertedLS := TIIB[RTDSK0-MPA-EL1008]^Channel 5^Input;
                             .i_xRetractedLS := TIIB[RTDSK0-MPA-EL1008]^Channel 6^Input;
                             .q_xInsert_DO :=  TIIB[RTDSK0-MPA-EL2008]^Channel 5^Output;
                             .q_xRetract_DO :=  TIIB[RTDSK0-MPA-EL2008]^Channel 6^Output
    '}

    {attribute 'pytmc' :=' pv: RTDSK0:MPA:03 '}
    RTDSK0_MPA_03: FB_MPA := (sName := 'RTDSK0:MPA:03');

       {attribute 'TcLinkTo' := '.i_xInsertedLS := TIIB[RTDSK0-MPA-EL1008]^Channel 7^Input;
                             .i_xRetractedLS := TIIB[RTDSK0-MPA-EL1008]^Channel 8^Input;
                             .q_xInsert_DO :=  TIIB[RTDSK0-MPA-EL2008]^Channel 7^Output;
                             .q_xRetract_DO :=  TIIB[RTDSK0-MPA-EL2008]^Channel 8^Output
    '}
    {attribute 'pytmc' :=' pv: RTDSK0:MPA:04 '}
    RTDSK0_MPA_04: FB_MPA := (sName := 'RTDSK0:MPA:04');

    fbRTDSK0_SCRP_MMS_Z: FB_MotionStage;
    fbRTDSK0_SCRP_MMS_X: FB_MotionStage;
    fbRTDSK0_SCRP_MMS_Y: FB_MotionStage;

     {attribute 'pytmc' := 'pv: RTDSK0:SCRP:LED:01:PWR
      io: io
        field: ZNAM OFF
        field: ONAM ON
'}

     {attribute 'TcLinkTo' := 'TIIB[RTDSK0-EL2004]^Channel 3^Output'}
    bRTDSK0_SCRP_LED_01 AT %Q*: BOOL;

    FFO : FB_FastFault :=( i_Desc := 'fault occurs when Y motor is not activating upper limit switch', i_TypeCode := 16#FAF, i_DevName := 'RTDSK0:SCRP:MMS:Y');
    bInit: BOOL := TRUE;



END_VAR


//Pneumatic actuators - OTR filters

RTDSK0_MPA_01(
    ibInsertOK:= TRUE,
    ibRetractOK:= TRUE ,
    ibPMPS_OK:= TRUE ,
    ibOverrideInterlock:= ,
    q_stAct=> ,
    xMPS_OK=> ,
    xDone=> ,
    i_xReset := ,
    io_fbFFHWO := GVL.fbFastFaultOutput1,
);

RTDSK0_MPA_02(
    ibInsertOK:= TRUE,
    ibRetractOK:= TRUE ,
    ibPMPS_OK:= TRUE ,
    ibOverrideInterlock:= ,
    q_stAct=> ,
    xMPS_OK=> ,
    xDone=> ,
    i_xReset := ,
    io_fbFFHWO := GVL.fbFastFaultOutput1,
);

(*
Disable MPA_03 and MPA_04, no actuator installed

RTDSK0_MPA_03(
    ibInsertOK:= TRUE,
    ibRetractOK:= TRUE ,
    ibPMPS_OK:= TRUE ,
    ibOverrideInterlock:= ,
    q_stAct=> ,
    xMPS_OK=> ,
    xDone=> ,
    i_xReset := ,
    io_fbFFHWO := GVL.fbFastFaultOutput1,
);

RTDSK0_MPA_04(
    ibInsertOK:= TRUE,
    ibRetractOK:= TRUE ,
    ibPMPS_OK:= TRUE ,
    ibOverrideInterlock:= ,
    q_stAct=> ,
    xMPS_OK=> ,
    xDone=> ,
    i_xReset := ,
    io_fbFFHWO := GVL.fbFastFaultOutput1,
);
*)

//initialize RTDSK0 stages
IF bInit THEN
    Main.M11.bHardwareEnable := TRUE;
    Main.M11.bPowerSelf :=TRUE;
    Main.M11.nBrakeMode := ENUM_StageBrakeMode.NO_BRAKE;
    Main.M11.nEnableMode := ENUM_StageEnableMode.DURING_MOTION;
    Main.M11.fHomePosition := 0;

    Main.M12.bHardwareEnable := TRUE;
    Main.M12.bPowerSelf :=TRUE;
    Main.M12.nBrakeMode := ENUM_StageBrakeMode.NO_BRAKE;
    Main.M12.nEnableMode := ENUM_StageEnableMode.DURING_MOTION;
    Main.M12.fHomePosition := 0;

    Main.M13.bHardwareEnable := TRUE;
    Main.M13.bPowerSelf :=TRUE;
    Main.M13.nBrakeMode := ENUM_StageBrakeMode.NO_BRAKE;
    Main.M13.nEnableMode := ENUM_StageEnableMode.DURING_MOTION;
    Main.M13.fHomePosition := 0;

    Main.M11.nHomingMode := ENUM_EpicsHomeCmd.HIGH_LIMIT;
    Main.M12.nHomingMode := ENUM_EpicsHomeCmd.HIGH_LIMIT;
    Main.M13.nHomingMode := ENUM_EpicsHomeCmd.HIGH_LIMIT;

    bInit := FALSE;
END_IF

    fbRTDSK0_SCRP_MMS_Z (stMotionStage := Main.M11);
    fbRTDSK0_SCRP_MMS_X (stMotionStage := Main.M12);
    fbRTDSK0_SCRP_MMS_Y (stMotionStage := Main.M13);
    FFO(i_xOK := NOT(Main.M13.bLimitForwardEnable) AND Main.M13.bLimitBackwardEnable, io_fbFFHWO := GVL.fbFastFaultOutput1);

END_PROGRAM

// ---- POUs/PRG_SL1K0_POWER.TcPOU
PROGRAM PRG_SL1K0_POWER
VAR
    {attribute 'pytmc' := '
        pv: SL1K0:POWER
        io: io
    '}
    {attribute 'TcLinkTo' := '.RTD_South_1.iRaw := TIIB[SL1K0-EL3202-E6]^RTD Inputs Channel 1^Value;
                              .RTD_South_1.bError := TIIB[SL1K0-EL3202-E6]^RTD Inputs Channel 1^Status^Error;
                              .RTD_South_1.bUnderrange := TIIB[SL1K0-EL3202-E6]^RTD Inputs Channel 1^Status^Underrange;
                              .RTD_South_1.bOverrange := TIIB[SL1K0-EL3202-E6]^RTD Inputs Channel 1^Status^Overrange;
                              .RTD_South_2.iRaw := TIIB[SL1K0-EL3202-E6]^RTD Inputs Channel 2^Value;
                              .RTD_South_2.bError := TIIB[SL1K0-EL3202-E6]^RTD Inputs Channel 2^Status^Error;
                              .RTD_South_2.bUnderrange := TIIB[SL1K0-EL3202-E6]^RTD Inputs Channel 2^Status^Underrange;
                              .RTD_South_2.bOverrange := TIIB[SL1K0-EL3202-E6]^RTD Inputs Channel 2^Status^Overrange;
                              .RTD_TOP_1.iRaw := TIIB[SL1K0-EL3202-E7]^RTD Inputs Channel 1^Value;
                              .RTD_TOP_1.bError := TIIB[SL1K0-EL3202-E7]^RTD Inputs Channel 1^Status^Error;
                              .RTD_TOP_1.bUnderrange := TIIB[SL1K0-EL3202-E7]^RTD Inputs Channel 1^Status^Underrange;
                              .RTD_TOP_1.bOverrange := TIIB[SL1K0-EL3202-E7]^RTD Inputs Channel 1^Status^Overrange;
                              .RTD_TOP_2.iRaw := TIIB[SL1K0-EL3202-E7]^RTD Inputs Channel 2^Value;
                              .RTD_TOP_2.bError := TIIB[SL1K0-EL3202-E7]^RTD Inputs Channel 2^Status^Error;
                              .RTD_TOP_2.bUnderrange := TIIB[SL1K0-EL3202-E7]^RTD Inputs Channel 2^Status^Underrange;
                              .RTD_TOP_2.bOverrange := TIIB[SL1K0-EL3202-E7]^RTD Inputs Channel 2^Status^Overrange;
                              .RTD_North_1.iRaw := TIIB[SL1K0-EL3202-E8]^RTD Inputs Channel 1^Value;
                              .RTD_North_1.bError := TIIB[SL1K0-EL3202-E8]^RTD Inputs Channel 1^Status^Error;
                              .RTD_North_1.bUnderrange := TIIB[SL1K0-EL3202-E8]^RTD Inputs Channel 1^Status^Underrange;
                              .RTD_North_1.bOverrange := TIIB[SL1K0-EL3202-E8]^RTD Inputs Channel 1^Status^Overrange;
                              .RTD_North_2.iRaw := TIIB[SL1K0-EL3202-E8]^RTD Inputs Channel 2^Value;
                              .RTD_North_2.bError := TIIB[SL1K0-EL3202-E8]^RTD Inputs Channel 2^Status^Error;
                              .RTD_North_2.bUnderrange := TIIB[SL1K0-EL3202-E8]^RTD Inputs Channel 2^Status^Underrange;
                              .RTD_North_2.bOverrange := TIIB[SL1K0-EL3202-E8]^RTD Inputs Channel 2^Status^Overrange;
                              .RTD_Bottom_1.iRaw := TIIB[SL1K0-EL3202-E9]^RTD Inputs Channel 1^Value;
                              .RTD_Bottom_1.bError := TIIB[SL1K0-EL3202-E9]^RTD Inputs Channel 1^Status^Error;
                              .RTD_Bottom_1.bUnderrange := TIIB[SL1K0-EL3202-E9]^RTD Inputs Channel 1^Status^Underrange;
                              .RTD_Bottom_1.bOverrange := TIIB[SL1K0-EL3202-E9]^RTD Inputs Channel 1^Status^Overrange;
                              .RTD_Bottom_2.iRaw := TIIB[SL1K0-EL3202-E9]^RTD Inputs Channel 2^Value;
                              .RTD_Bottom_2.bError := TIIB[SL1K0-EL3202-E9]^RTD Inputs Channel 2^Status^Error;
                              .RTD_Bottom_2.bUnderrange := TIIB[SL1K0-EL3202-E9]^RTD Inputs Channel 2^Status^Underrange;
                              .RTD_Bottom_2.bOverrange := TIIB[SL1K0-EL3202-E9]^RTD Inputs Channel 2^Status^Overrange;
                              .AptArrayStatus := TIIB[PMPS_PRE]^IO Outputs^AptArrayStatus^AptArrayStatus[1];
                              .AptArrayReq := TIIB[PMPS_PRE]^IO Inputs^AptArrayReq^AptArrayReq[1];
                              .fbFlowSwitch.bFlowOk := TIIB[IM1K0-EL1004]^Channel 3^Input'}
    fbSL1K0: FB_SLITS_POWER;
//{attribute 'TcLinkTo' := 'TIIB[PMPS_PRE]^IO Outputs^AptArrayStatus'}
    {attribute 'pytmc' := '
    pv: SL1K0:POWER:GO;
    io: io;
    field: ZNAM False;
    field: ONAM True;
    '}
    bExecuteMotion:BOOL ;
    //GET PMPS Move Ok bit
    // Default True until it is properly linked to PMPS bit
    bMoveOk:BOOL :=TRUE;

    //for testing purposes only. comment-out/delete once done.
    mcPower : ARRAY [1..4] OF MC_POWER;
    bTest:BOOL:=FALSE;

    (*Offsets*)
    (* Absolute encoder value at the HLS + Absolure eoncoder value at the centered beam *)
    rEncoderOffsetTop: REAL :=  -11.2; // -11.810; (* 0+(-15)*)
    rEncoderOffsetBottom: REAL := -12.02; //-12.499; (* 0+(-15)*)
    rEncoderOffsetNorth: REAL := -10.88; // -11.4;//-4.6;(* 0+(-15)*)
    rEncoderOffsetSouth: REAL := -12.475; //-13;(* 0+(-15)*)
END_VAR


fbSL1K0.bMoveOk := bMoveOk;
Main.M18.bLimitBackwardEnable := True;



//for testing purposes only. comment-out/delete once done.
If bTest THEN
    mcPower[1](axis:=Main.M18.Axis, Enable:=TRUE, enable_positive:=Main.M18.bLimitForwardEnable, enable_negative:=Main.M18.bLimitBackwardEnable);
mcPower[2](axis:=Main.M19.Axis, Enable:=TRUE, enable_positive:=Main.M19.bLimitForwardEnable, enable_negative:=Main.M19.bLimitBackwardEnable);
mcPower[3](axis:=Main.M20.Axis, Enable:=TRUE, enable_positive:=Main.M20.bLimitForwardEnable, enable_negative:=Main.M20.bLimitBackwardEnable);
mcPower[4](axis:=Main.M21.Axis, Enable:=TRUE, enable_positive:=Main.M21.bLimitForwardEnable, enable_negative:=Main.M21.bLimitBackwardEnable);

else

//force that inner limit switch on south motor is not depressed. need to debug further in winter down.
//Main.M18.bLimitForwardEnable := TRUE;
fbSL1K0.rEncoderOffsetTop := rEncoderOffsetTop;
fbSL1K0.rEncoderOffsetBottom := rEncoderOffsetBottom;
fbSL1K0.rEncoderOffsetNorth := rEncoderOffsetNorth;
fbSL1K0.rEncoderOffsetSouth := rEncoderOffsetSouth;

fbSL1K0(stTopBlade:=  Main.M19,
        stBottomBlade:= Main.M21,
        stNorthBlade:=  Main.M20,
        stSouthBlade:=  Main.M18,
        bExecuteMotion:=bExecuteMotion,
        io_fbFFHWO := GVL.fbFastFaultOutput1,
        fbArbiter := GVL.fbArbiter);

fbSL1K0.M_UpdatePMPS(1);

END_IF

END_PROGRAM

// ---- Temp/FB_SLITS_POWER.TcPOU
FUNCTION_BLOCK FB_SLITS_POWER EXTENDS FB_SLITS
VAR_INPUT
END_VAR
VAR
    {attribute 'pytmc' := '
    pv: MODE ;
     field: ZNAM Local;
    field: ONAM PMPS;
     io: io;
    '}
    xPMPSMode	:BOOL :=TRUE;


     {attribute 'pytmc' := '
        pv: FSW
    '}
    fbFlowSwitch: FB_XTES_Flowswitch;


    //RTDs
    {attribute 'pytmc' := '
        pv: TOP:RTD:01
    '}
    RTD_TOP_1: FB_TempSensor;
    {attribute 'pytmc' := '
        pv: TOP:RTD:02
    '}
    RTD_TOP_2: FB_TempSensor;
    {attribute 'pytmc' := '
        pv: BOTTOM:RTD:01
    '}
    RTD_Bottom_1: FB_TempSensor;
    {attribute 'pytmc' := '
        pv: BOTTOM:RTD:02
    '}
    RTD_Bottom_2: FB_TempSensor;

    {attribute 'pytmc' := '
        pv: NORTH:RTD:01
    '}
    RTD_North_1: FB_TempSensor;
    {attribute 'pytmc' := '
        pv: NORTH:RTD:02
    '}
    RTD_North_2: FB_TempSensor;
    {attribute 'pytmc' := '
        pv: SOUTH:RTD:01
    '}
    RTD_South_1: FB_TempSensor;
    {attribute 'pytmc' := '
        pv: SOUTH:RTD:02
    '}
    RTD_South_2: FB_TempSensor;


END_VAR

ACT_init();

// Instantiate Function block for all the blades
ACT_Motion();
//SET and GET the requested and Actual values
ACT_CalculatePositions();
//ACT_BLOCK();
ACT_RTDs();

ACTION ACT_RTDs:
////RTDs
RTD_TOP_1();
RTD_TOP_2();
RTD_Bottom_1();
RTD_Bottom_2();
RTD_North_1();
RTD_North_2();
RTD_South_1();
RTD_South_2();

//Flow Switch
fbFlowSwitch();
END_ACTION

METHOD M_UpdatePMPS : BOOL
VAR_INPUT
    index: int;
END_VAR
//Keep updating the status of the apertures PMPS
This^.AptArrayStatus.Height := This^.rActApertureSizeY;
This^.AptArrayStatus.Width := This^.rActApertureSizeX;
This^.AptArrayStatus.xOK := NOT (This^.stTopBlade.bError) AND NOT (This^.stBottomBlade.bError)
                                 AND NOT (This^.stNorthBlade.bError) AND NOT (This^.stNorthBlade.bError);

//Evaluate that the current center on the X and the y direction didn't exceed limits,
// Gap should be reduced when center is moved, gap < Maximum permessible gap - 2|Center deviation from nominal|
//Fast fault when it does.
IF(This^.rActApertureSizeX > (AptArrayReq.Width - (2*ABS(rActCenterX)))
//(rActCenterX > (PMPS_GVL.stCurrentBeamParameters.astApertures[index].Width/2))
    AND (PMPS_GVL.stCurrentBeamParameters.astApertures[index].Width >0 ))
    OR (This^.rActApertureSizeY > (AptArrayReq.Height - (2*ABS(rActCenterY)))
    //((rActCenterY > (PMPS_GVL.stCurrentBeamParameters.astApertures[index].Height/2))
        AND(PMPS_GVL.stCurrentBeamParameters.astApertures[index].Height>0 )) THEN
        FFO.i_xOK := FALSE;
    ELSE
        FFO.i_xOK := TRUE;
END_IF

//Evaluate that the requested gaps on the X and the y direction is not larger than the current gap
// narrow  the gap if the requested is larger
IF(xPMPSMode) THEN
    IF (This^.rActApertureSizeX > AptArrayReq.Width) THEN
        rReqApertureSizeX := AptArrayReq.Width - 0.01;
    END_IF
    IF (This^.rActApertureSizeY > AptArrayReq.Height) THEN
         rReqApertureSizeY := AptArrayReq.Height - 0.01;
    END_IF
    ELSE
     FFO.i_xOK := FALSE;
END_IF


(*FAST FAULT*)
FFO(i_xOK := ,
    i_xReset := ,
    i_xAutoReset :=TRUE,
    io_fbFFHWO := io_fbFFHWO);
END_METHOD

END_FUNCTION_BLOCK

// ---- Temp/FB_SLITS.TcPOU
FUNCTION_BLOCK FB_SLITS
VAR_IN_OUT
    stTopBlade: ST_MotionStage;
    stBottomBlade: ST_MotionStage;
    stNorthBlade: ST_MotionStage;
    stSouthBlade: ST_MotionStage;
    bExecuteMotion:BOOL ;
    io_fbFFHWO    :    FB_HardwareFFOutput;
    fbArbiter: FB_Arbiter();
END_VAR

VAR_INPUT

    {attribute 'pytmc' := '
    pv: PMPS_OK;
    io: i;
    field: ZNAM False
    field: ONAM True
    '}
    bMoveOk:BOOL;

        (*Offsets*)
    {attribute 'pytmc' := '
    pv: Offset_Top;
    io: io;
    '}
    rEncoderOffsetTop: REAL;
    {attribute 'pytmc' := '
    pv: ZeroOffset_Bottom;
    io: io;
    '}
    rEncoderOffsetBottom: REAL;
    {attribute 'pytmc' := '
    pv: ZeroOffset_North;
    io: io;
    '}
    rEncoderOffsetNorth: REAL;
    {attribute 'pytmc' := '
    pv: ZeroOffset_South;
    io: io;
    '}
    rEncoderOffsetSouth: REAL;
    i_DevName : STRING; //device name for FFO and PMPS diagnostics
END_VAR

VAR
    fbTopBlade: FB_MotionStage;
    fbBottomBlade: FB_MotionStage;
    fbNorthBlade: FB_MotionStage;
    fbSouthBlade: FB_MotionStage;
    fPosTopBlade: LREAL;
    fPosBottomBlade: LREAL;
    fPosNorthBlade: LREAL;
    fPosSouthBlade: LREAL;

    (*Motion Parameters*)
    fSmallDelta: LREAL := 0.01;
    fBigDelta: LREAL := 10;
    fMaxVelocity: LREAL := 0.2;
    fHighAccel: LREAL := 0.8;
    fLowAccel: LREAL := 0.1;

    stTop: DUT_PositionState;
    stBOTTOM: DUT_PositionState;
    stNorth: DUT_PositionState;
    stSouth: DUT_PositionState;

    {attribute 'pytmc' := 'pv: TOP'}
    fbTop: FB_StatePTPMove;
    {attribute 'pytmc' := 'pv: BOTTOM'}
    fbBottom: FB_StatePTPMove;
    {attribute 'pytmc' := 'pv: NORTH'}
    fbNorth: FB_StatePTPMove;
    {attribute 'pytmc' := 'pv: SOUTH'}
    fbSouth: FB_StatePTPMove;

    (*EPICS pvs*)
    {attribute 'pytmc' := '
    pv: XWID_REQ;
    io: io;
    '}
    rReqApertureSizeX : REAL;
    {attribute 'pytmc' := '
    pv: YWID_REQ;
    io: io;
    '}
    rReqApertureSizeY : REAL;
    {attribute 'pytmc' := '
    pv: XCEN_REQ;
    io: io;
    '}
    rReqCenterX: REAL;
    {attribute 'pytmc' := '
    pv: YCEN_REQ;
    io: io;
    '}
    rReqCenterY: REAL;

